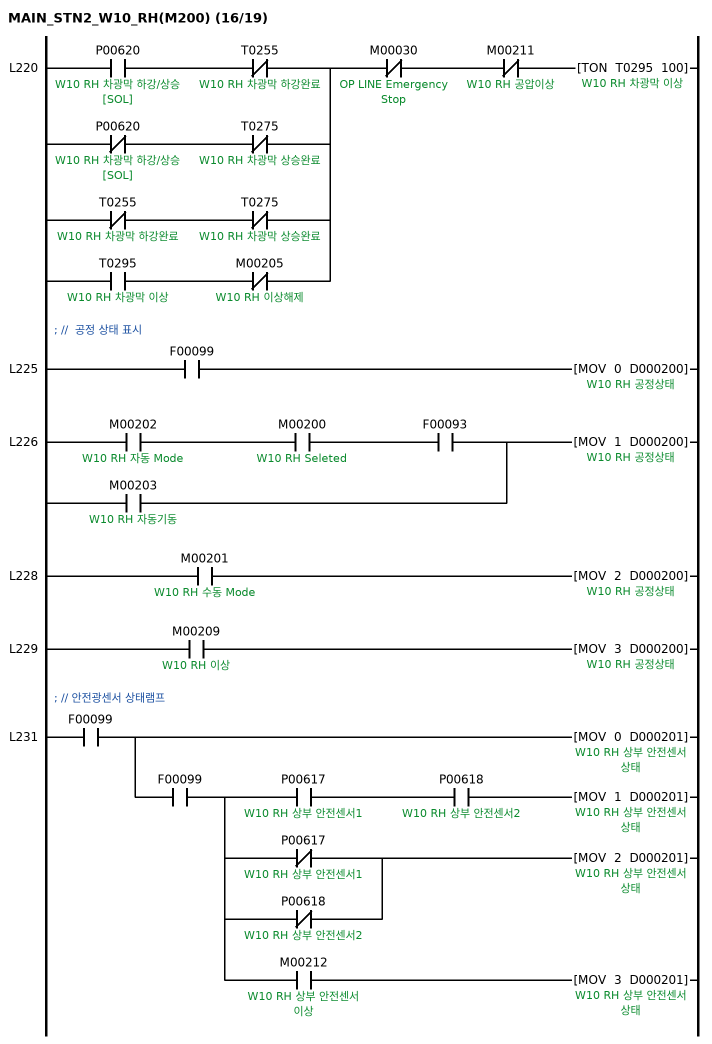
[picture p72: MAIN_STN2_W10_RH(M200) rungs L220-L231]
; L220
LOAD      P00620	// W10 RH 차광막 하강/상승 [SOL]
AND NOT   T0255	// W10 RH 차광막 하강완료
LOAD NOT  P00620	// W10 RH 차광막 하강/상승 [SOL]
AND NOT   T0275	// W10 RH 차광막 상승완료
OR LOAD
LOAD NOT  T0255	// W10 RH 차광막 하강완료
AND NOT   T0275	// W10 RH 차광막 상승완료
OR LOAD
LOAD      T0295	// W10 RH 차광막 이상
AND NOT   M00205	// W10 RH 이상해제
OR LOAD
AND NOT   M00030	// OP LINE Emergency Stop
AND NOT   M00211	// W10 RH 공압이상
TON       T0295 100	// W10 RH 차광막 이상
//   //  공정 상태 표시
; L225
LOAD      F00099
MOV       0 D000200	// W10 RH 공정상태
; L226
LOAD      M00202	// W10 RH 자동 Mode
AND       M00200	// W10 RH Seleted
AND       F00093
OR        M00203	// W10 RH 자동기동
MOV       1 D000200	// W10 RH 공정상태
; L228
LOAD      M00201	// W10 RH 수동 Mode
MOV       2 D000200	// W10 RH 공정상태
; L229
LOAD      M00209	// W10 RH 이상
MOV       3 D000200	// W10 RH 공정상태
//   // 안전광센서 상태램프
; L231
LOAD      F00099
MOV       0 D000201	// W10 RH 상부 안전센서 상태
AND       F00099
MPUSH
AND       P00617	// W10 RH 상부 안전센서1
AND       P00618	// W10 RH 상부 안전센서2
MOV       1 D000201	// W10 RH 상부 안전센서 상태
MLOAD
LOAD NOT  P00617	// W10 RH 상부 안전센서1
OR NOT    P00618	// W10 RH 상부 안전센서2
AND LOAD
MOV       2 D000201	// W10 RH 상부 안전센서 상태
MPOP
AND       M00212	// W10 RH 상부 안전센서 이상
MOV       3 D000201	// W10 RH 상부 안전센서 상태

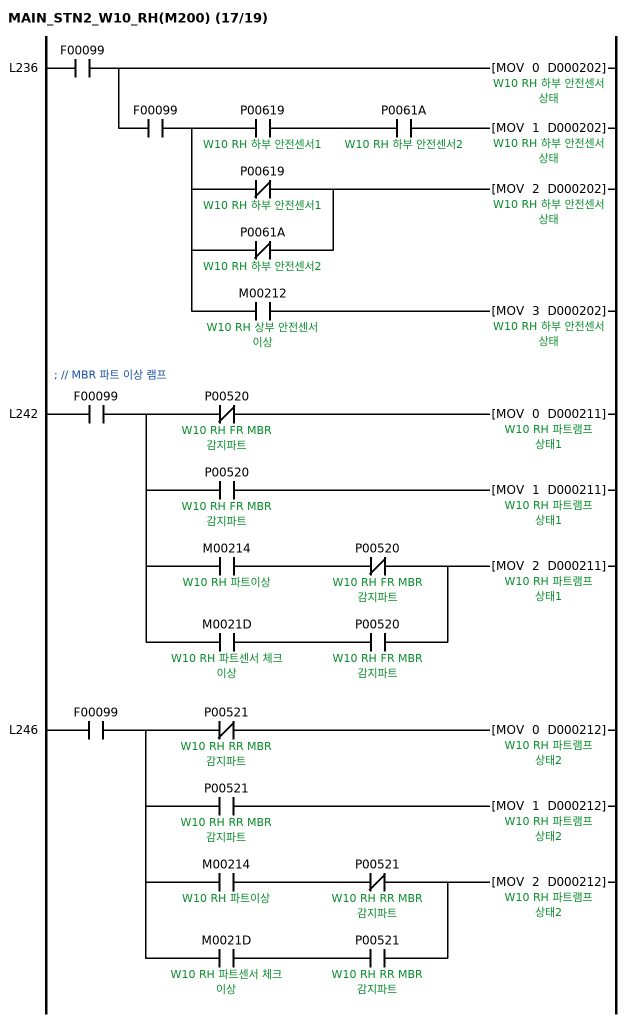
; L236
LOAD      F00099
MOV       0 D000202	// W10 RH 하부 안전센서 상태
AND       F00099
MPUSH
AND       P00619	// W10 RH 하부 안전센서1
AND       P0061A	// W10 RH 하부 안전센서2
MOV       1 D000202	// W10 RH 하부 안전센서 상태
MLOAD
LOAD NOT  P00619	// W10 RH 하부 안전센서1
OR NOT    P0061A	// W10 RH 하부 안전센서2
AND LOAD
MOV       2 D000202	// W10 RH 하부 안전센서 상태
MPOP
AND       M00212	// W10 RH 상부 안전센서 이상
MOV       3 D000202	// W10 RH 하부 안전센서 상태
//   // MBR 파트 이상 램프
; L242
LOAD      F00099
MPUSH
AND NOT   P00520	// W10 RH FR MBR 감지파트
MOV       0 D000211	// W10 RH 파트램프 상태1
MLOAD
AND       P00520	// W10 RH FR MBR 감지파트
MOV       1 D000211	// W10 RH 파트램프 상태1
MPOP
LOAD      M00214	// W10 RH 파트이상
AND NOT   P00520	// W10 RH FR MBR 감지파트
LOAD      M0021D	// W10 RH 파트센서 체크 이상
AND       P00520	// W10 RH FR MBR 감지파트
OR LOAD
AND LOAD
MOV       2 D000211	// W10 RH 파트램프 상태1
; L246
LOAD      F00099
MPUSH
AND NOT   P00521	// W10 RH RR MBR 감지파트
MOV       0 D000212	// W10 RH 파트램프 상태2
MLOAD
AND       P00521	// W10 RH RR MBR 감지파트
MOV       1 D000212	// W10 RH 파트램프 상태2
MPOP
LOAD      M00214	// W10 RH 파트이상
AND NOT   P00521	// W10 RH RR MBR 감지파트
LOAD      M0021D	// W10 RH 파트센서 체크 이상
AND       P00521	// W10 RH RR MBR 감지파트
OR LOAD
AND LOAD
MOV       2 D000212	// W10 RH 파트램프 상태2

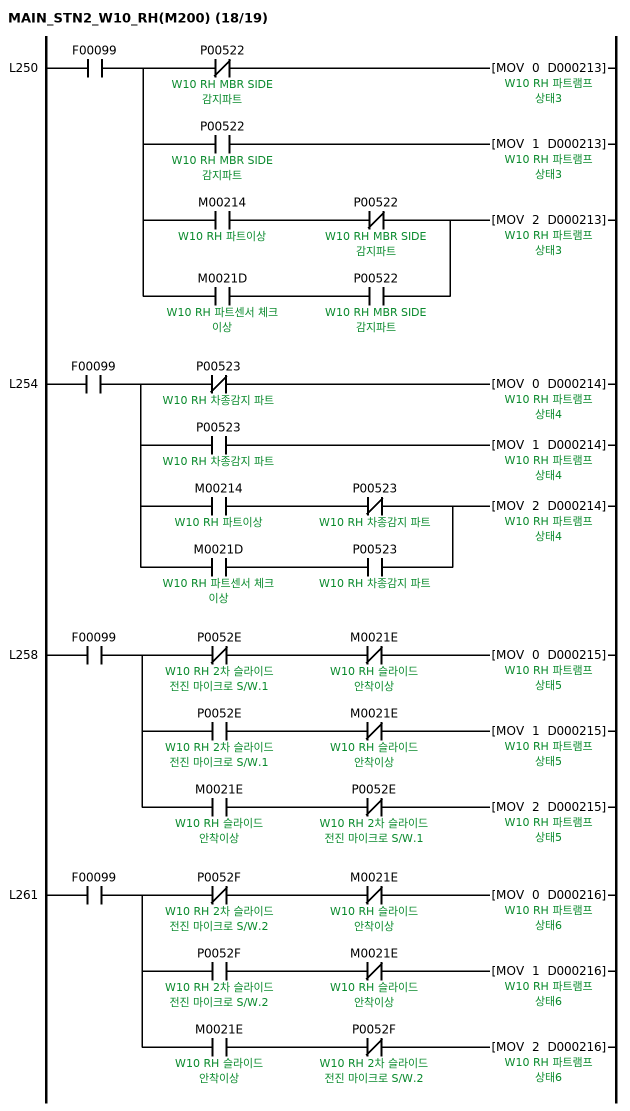
; L250
LOAD      F00099
MPUSH
AND NOT   P00522	// W10 RH MBR SIDE 감지파트
MOV       0 D000213	// W10 RH 파트램프 상태3
MLOAD
AND       P00522	// W10 RH MBR SIDE 감지파트
MOV       1 D000213	// W10 RH 파트램프 상태3
MPOP
LOAD      M00214	// W10 RH 파트이상
AND NOT   P00522	// W10 RH MBR SIDE 감지파트
LOAD      M0021D	// W10 RH 파트센서 체크 이상
AND       P00522	// W10 RH MBR SIDE 감지파트
OR LOAD
AND LOAD
MOV       2 D000213	// W10 RH 파트램프 상태3
; L254
LOAD      F00099
MPUSH
AND NOT   P00523	// W10 RH 차종감지 파트
MOV       0 D000214	// W10 RH 파트램프 상태4
MLOAD
AND       P00523	// W10 RH 차종감지 파트
MOV       1 D000214	// W10 RH 파트램프 상태4
MPOP
LOAD      M00214	// W10 RH 파트이상
AND NOT   P00523	// W10 RH 차종감지 파트
LOAD      M0021D	// W10 RH 파트센서 체크 이상
AND       P00523	// W10 RH 차종감지 파트
OR LOAD
AND LOAD
MOV       2 D000214	// W10 RH 파트램프 상태4
; L258
LOAD      F00099
MPUSH
AND NOT   P0052E	// W10 RH 2차 슬라이드 전진 마이크로 S/W.1
AND NOT   M0021E	// W10 RH 슬라이드 안착이상
MOV       0 D000215	// W10 RH 파트램프 상태5
MLOAD
AND       P0052E	// W10 RH 2차 슬라이드 전진 마이크로 S/W.1
AND NOT   M0021E	// W10 RH 슬라이드 안착이상
MOV       1 D000215	// W10 RH 파트램프 상태5
MPOP
AND       M0021E	// W10 RH 슬라이드 안착이상
AND NOT   P0052E	// W10 RH 2차 슬라이드 전진 마이크로 S/W.1
MOV       2 D000215	// W10 RH 파트램프 상태5
; L261
LOAD      F00099
MPUSH
AND NOT   P0052F	// W10 RH 2차 슬라이드 전진 마이크로 S/W.2
AND NOT   M0021E	// W10 RH 슬라이드 안착이상
MOV       0 D000216	// W10 RH 파트램프 상태6
MLOAD
AND       P0052F	// W10 RH 2차 슬라이드 전진 마이크로 S/W.2
AND NOT   M0021E	// W10 RH 슬라이드 안착이상
MOV       1 D000216	// W10 RH 파트램프 상태6
MPOP
AND       M0021E	// W10 RH 슬라이드 안착이상
AND NOT   P0052F	// W10 RH 2차 슬라이드 전진 마이크로 S/W.2
MOV       2 D000216	// W10 RH 파트램프 상태6

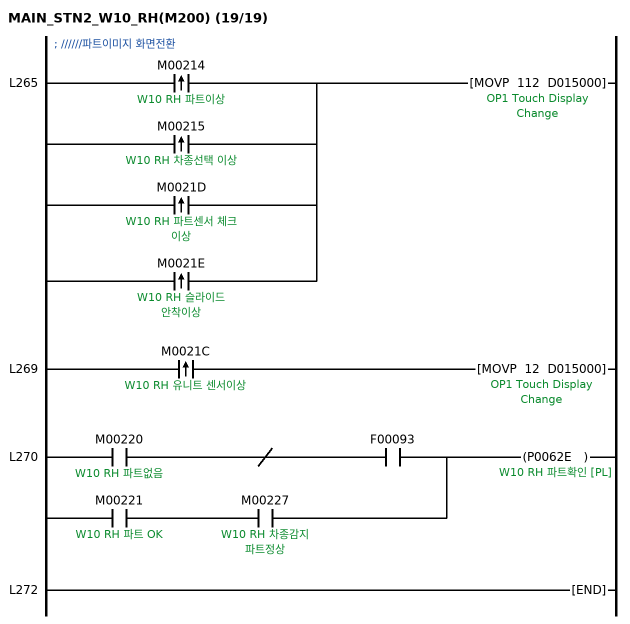
// //////파트이미지 화면전환
; L265
LOADP     M00214	// W10 RH 파트이상
ORP       M00215	// W10 RH 차종선택 이상
ORP       M0021D	// W10 RH 파트센서 체크 이상
ORP       M0021E	// W10 RH 슬라이드 안착이상
MOVP      112 D015000	// OP1 Touch Display Change
; L269
LOADP     M0021C	// W10 RH 유니트 센서이상
MOVP      12 D015000	// OP1 Touch Display Change
; L270
LOAD      M00220	// W10 RH 파트없음
NOT
AND       F00093
LOAD      M00221	// W10 RH 파트 OK
AND       M00227	// W10 RH 차종감지 파트정상
OR LOAD
OUT       P0062E	// W10 RH 파트확인 [PL]
; L272
END

PROGRAM MAIN_STN3_W20_LH_냉각(M300) (task: 스캔 프로그램)

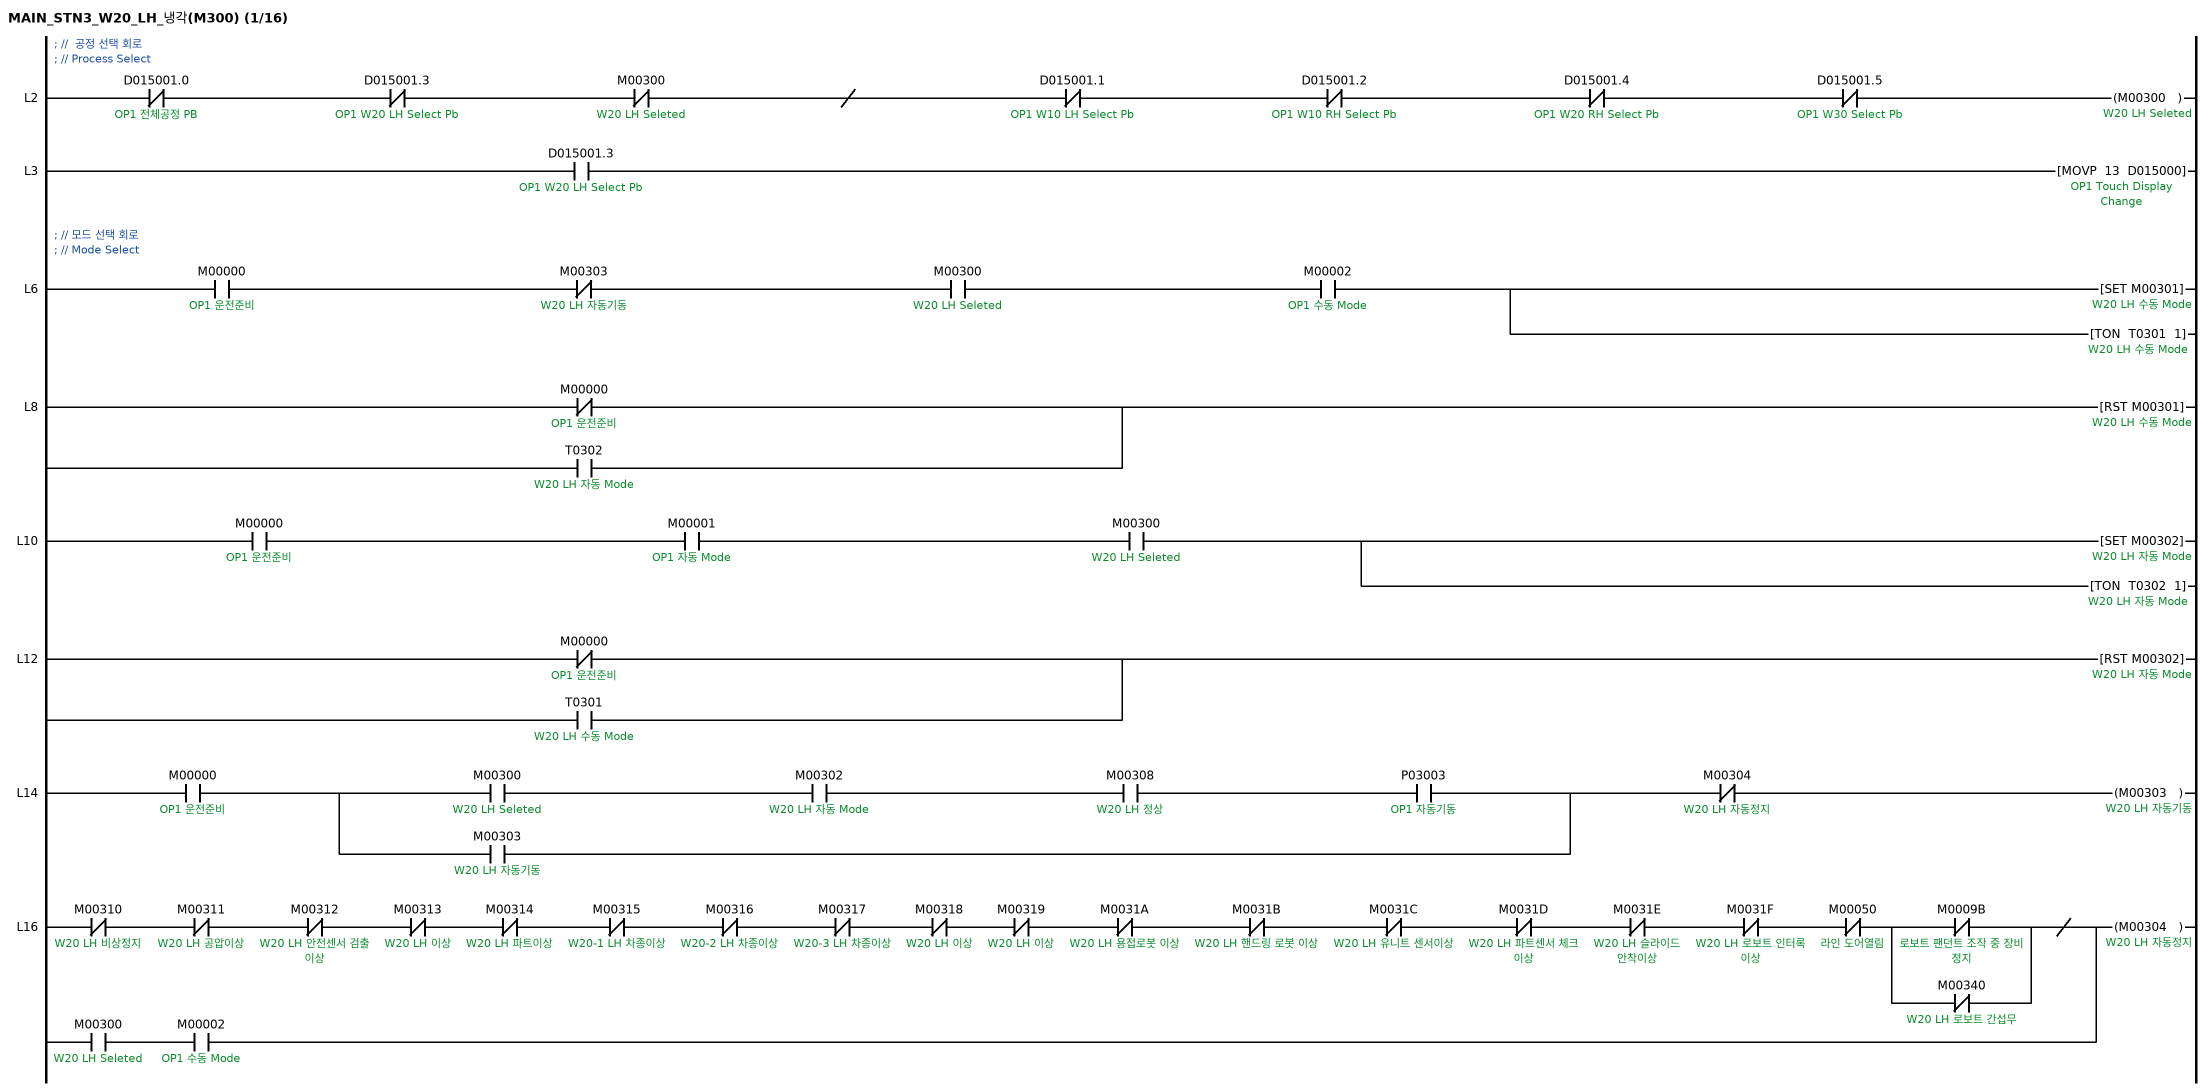
//   //  공정 선택 회로
//   // Process Select
; L2
LOAD NOT  D015001.0	// OP1 전체공정 PB
AND NOT   D015001.3	// OP1 W20 LH Select Pb
AND NOT   M00300	// W20 LH Seleted
NOT
AND NOT   D015001.1	// OP1 W10 LH Select Pb
AND NOT   D015001.2	// OP1 W10 RH Select Pb
AND NOT   D015001.4	// OP1 W20 RH Select Pb
AND NOT   D015001.5	// OP1 W30 Select Pb
OUT       M00300	// W20 LH Seleted
; L3
LOAD      D015001.3	// OP1 W20 LH Select Pb
MOVP      13 D015000	// OP1 Touch Display Change
// // 모드 선택 회로
//   // Mode Select
; L6
LOAD      M00000	// OP1 운전준비
AND NOT   M00303	// W20 LH 자동기동
AND       M00300	// W20 LH Seleted
AND       M00002	// OP1 수동 Mode
SET       M00301	// W20 LH 수동 Mode
TON       T0301 1	// W20 LH 수동 Mode
; L8
LOAD NOT  M00000	// OP1 운전준비
OR        T0302	// W20 LH 자동 Mode
RST       M00301	// W20 LH 수동 Mode
; L10
LOAD      M00000	// OP1 운전준비
AND       M00001	// OP1 자동 Mode
AND       M00300	// W20 LH Seleted
SET       M00302	// W20 LH 자동 Mode
TON       T0302 1	// W20 LH 자동 Mode
; L12
LOAD NOT  M00000	// OP1 운전준비
OR        T0301	// W20 LH 수동 Mode
RST       M00302	// W20 LH 자동 Mode
; L14
LOAD      M00000	// OP1 운전준비
LOAD      M00300	// W20 LH Seleted
AND       M00302	// W20 LH 자동 Mode
AND       M00308	// W20 LH 정상
AND       P03003	// OP1 자동기동
OR        M00303	// W20 LH 자동기동
AND LOAD
AND NOT   M00304	// W20 LH 자동정지
OUT       M00303	// W20 LH 자동기동
; L16
LOAD NOT  M00310	// W20 LH 비상정지
AND NOT   M00311	// W20 LH 공압이상
AND NOT   M00312	// W20 LH 안전센서 검출 이상
AND NOT   M00313	// W20 LH 이상
AND NOT   M00314	// W20 LH 파트이상
AND NOT   M00315	// W20-1 LH 차종이상
AND NOT   M00316	// W20-2 LH 차종이상
AND NOT   M00317	// W20-3 LH 차종이상
AND NOT   M00318	// W20 LH 이상
AND NOT   M00319	// W20 LH 이상
AND NOT   M0031A	// W20 LH 용접로봇 이상
AND NOT   M0031B	// W20 LH 핸드링 로봇 이상
AND NOT   M0031C	// W20 LH 유니트 센서이상
AND NOT   M0031D	// W20 LH 파트센서 체크 이상
AND NOT   M0031E	// W20 LH 슬라이드 안착이상
AND NOT   M0031F	// W20 LH 로보트 인터록 이상
AND NOT   M00050	// 라인 도어열림
LOAD NOT  M0009B	// 로보트 팬던트 조작 중 장비 정지
OR NOT    M00340	// W20 LH 로보트 간섭무
AND LOAD
NOT
LOAD      M00300	// W20 LH Seleted
AND       M00002	// OP1 수동 Mode
OR LOAD
OUT       M00304	// W20 LH 자동정지

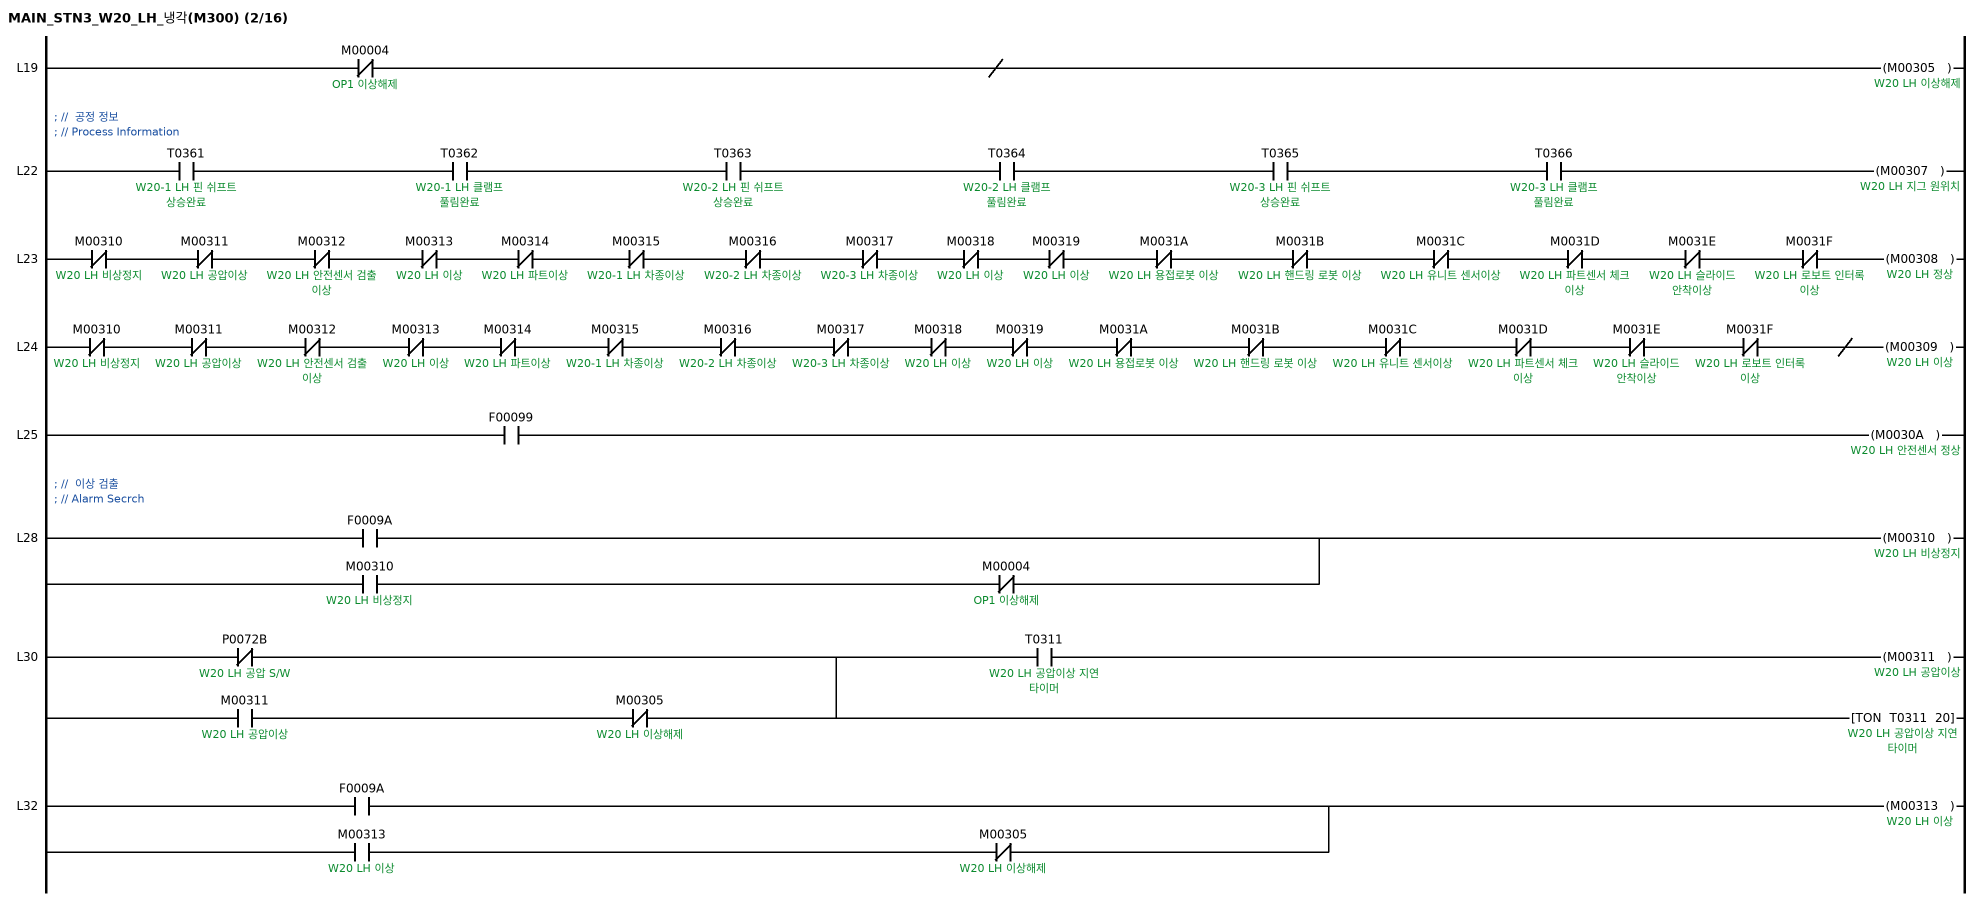
; L19
LOAD NOT  M00004	// OP1 이상해제
NOT
OUT       M00305	// W20 LH 이상해제
//   //  공정 정보
//   // Process Information
; L22
LOAD      T0361	// W20-1 LH 핀 쉬프트 상승완료
AND       T0362	// W20-1 LH 클램프 풀림완료
AND       T0363	// W20-2 LH 핀 쉬프트 상승완료
AND       T0364	// W20-2 LH 클램프 풀림완료
AND       T0365	// W20-3 LH 핀 쉬프트 상승완료
AND       T0366	// W20-3 LH 클램프 풀림완료
OUT       M00307	// W20 LH 지그 원위치
; L23
LOAD NOT  M00310	// W20 LH 비상정지
AND NOT   M00311	// W20 LH 공압이상
AND NOT   M00312	// W20 LH 안전센서 검출 이상
AND NOT   M00313	// W20 LH 이상
AND NOT   M00314	// W20 LH 파트이상
AND NOT   M00315	// W20-1 LH 차종이상
AND NOT   M00316	// W20-2 LH 차종이상
AND NOT   M00317	// W20-3 LH 차종이상
AND NOT   M00318	// W20 LH 이상
AND NOT   M00319	// W20 LH 이상
AND NOT   M0031A	// W20 LH 용접로봇 이상
AND NOT   M0031B	// W20 LH 핸드링 로봇 이상
AND NOT   M0031C	// W20 LH 유니트 센서이상
AND NOT   M0031D	// W20 LH 파트센서 체크 이상
AND NOT   M0031E	// W20 LH 슬라이드 안착이상
AND NOT   M0031F	// W20 LH 로보트 인터록 이상
OUT       M00308	// W20 LH 정상
; L24
LOAD NOT  M00310	// W20 LH 비상정지
AND NOT   M00311	// W20 LH 공압이상
AND NOT   M00312	// W20 LH 안전센서 검출 이상
AND NOT   M00313	// W20 LH 이상
AND NOT   M00314	// W20 LH 파트이상
AND NOT   M00315	// W20-1 LH 차종이상
AND NOT   M00316	// W20-2 LH 차종이상
AND NOT   M00317	// W20-3 LH 차종이상
AND NOT   M00318	// W20 LH 이상
AND NOT   M00319	// W20 LH 이상
AND NOT   M0031A	// W20 LH 용접로봇 이상
AND NOT   M0031B	// W20 LH 핸드링 로봇 이상
AND NOT   M0031C	// W20 LH 유니트 센서이상
AND NOT   M0031D	// W20 LH 파트센서 체크 이상
AND NOT   M0031E	// W20 LH 슬라이드 안착이상
AND NOT   M0031F	// W20 LH 로보트 인터록 이상
NOT
OUT       M00309	// W20 LH 이상
; L25
LOAD      F00099
OUT       M0030A	// W20 LH 안전센서 정상
//   //  이상 검출
//   // Alarm Secrch
; L28
LOAD      F0009A
LOAD      M00310	// W20 LH 비상정지
AND NOT   M00004	// OP1 이상해제
OR LOAD
OUT       M00310	// W20 LH 비상정지
; L30
LOAD NOT  P0072B	// W20 LH 공압 S/W
LOAD      M00311	// W20 LH 공압이상
AND NOT   M00305	// W20 LH 이상해제
OR LOAD
MPUSH
AND       T0311	// W20 LH 공압이상 지연 타이머
OUT       M00311	// W20 LH 공압이상
MPOP
TON       T0311 20	// W20 LH 공압이상 지연 타이머
; L32
LOAD      F0009A
LOAD      M00313	// W20 LH 이상
AND NOT   M00305	// W20 LH 이상해제
OR LOAD
OUT       M00313	// W20 LH 이상

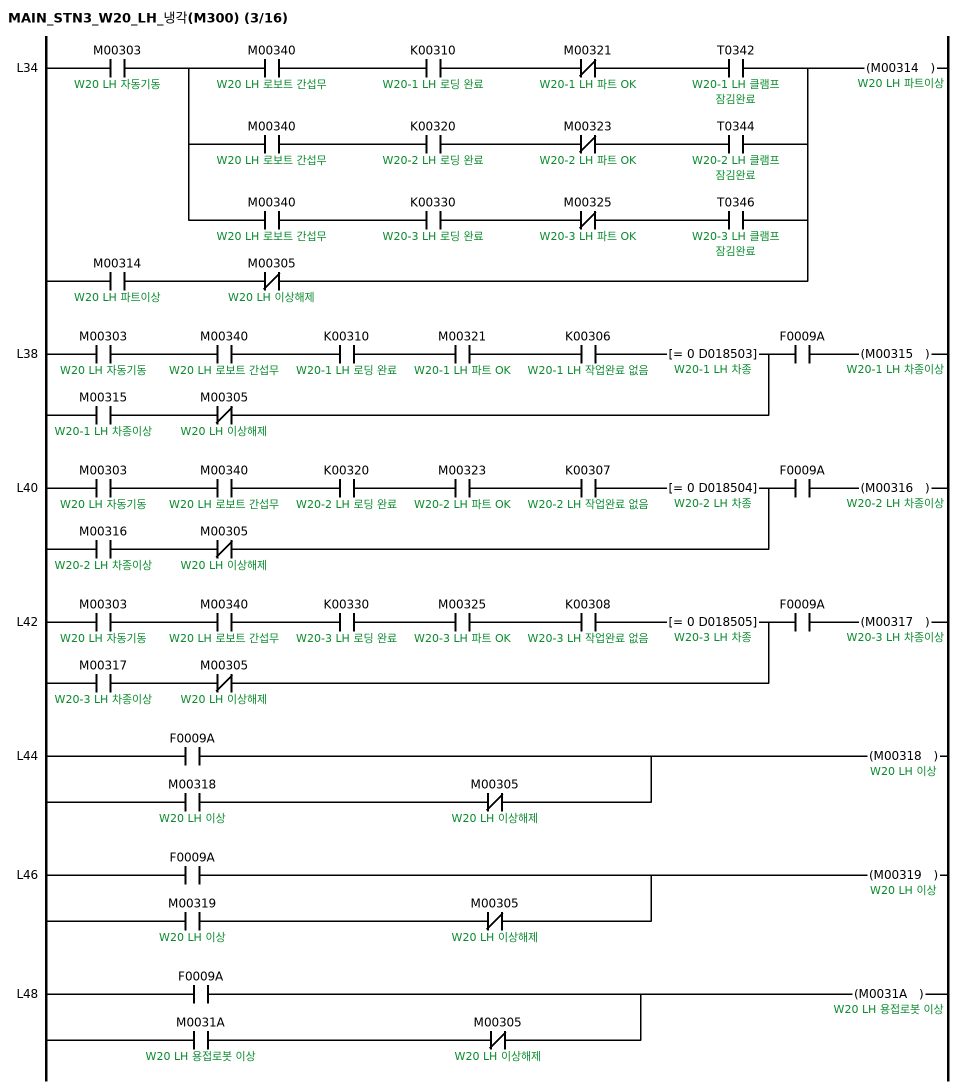
; L34
LOAD      M00303	// W20 LH 자동기동
LOAD      M00340	// W20 LH 로보트 간섭무
AND       K00310	// W20-1 LH 로딩 완료
AND NOT   M00321	// W20-1 LH 파트 OK
AND       T0342	// W20-1 LH 클램프 잠김완료
LOAD      M00340	// W20 LH 로보트 간섭무
AND       K00320	// W20-2 LH 로딩 완료
AND NOT   M00323	// W20-2 LH 파트 OK
AND       T0344	// W20-2 LH 클램프 잠김완료
OR LOAD
LOAD      M00340	// W20 LH 로보트 간섭무
AND       K00330	// W20-3 LH 로딩 완료
AND NOT   M00325	// W20-3 LH 파트 OK
AND       T0346	// W20-3 LH 클램프 잠김완료
OR LOAD
AND LOAD
LOAD      M00314	// W20 LH 파트이상
AND NOT   M00305	// W20 LH 이상해제
OR LOAD
OUT       M00314	// W20 LH 파트이상
; L38
LOAD      M00303	// W20 LH 자동기동
AND       M00340	// W20 LH 로보트 간섭무
AND       K00310	// W20-1 LH 로딩 완료
AND       M00321	// W20-1 LH 파트 OK
AND       K00306	// W20-1 LH 작업완료 없음
AND=      0 D018503	// W20-1 LH 차종
LOAD      M00315	// W20-1 LH 차종이상
AND NOT   M00305	// W20 LH 이상해제
OR LOAD
AND       F0009A
OUT       M00315	// W20-1 LH 차종이상
; L40
LOAD      M00303	// W20 LH 자동기동
AND       M00340	// W20 LH 로보트 간섭무
AND       K00320	// W20-2 LH 로딩 완료
AND       M00323	// W20-2 LH 파트 OK
AND       K00307	// W20-2 LH 작업완료 없음
AND=      0 D018504	// W20-2 LH 차종
LOAD      M00316	// W20-2 LH 차종이상
AND NOT   M00305	// W20 LH 이상해제
OR LOAD
AND       F0009A
OUT       M00316	// W20-2 LH 차종이상
; L42
LOAD      M00303	// W20 LH 자동기동
AND       M00340	// W20 LH 로보트 간섭무
AND       K00330	// W20-3 LH 로딩 완료
AND       M00325	// W20-3 LH 파트 OK
AND       K00308	// W20-3 LH 작업완료 없음
AND=      0 D018505	// W20-3 LH 차종
LOAD      M00317	// W20-3 LH 차종이상
AND NOT   M00305	// W20 LH 이상해제
OR LOAD
AND       F0009A
OUT       M00317	// W20-3 LH 차종이상
; L44
LOAD      F0009A
LOAD      M00318	// W20 LH 이상
AND NOT   M00305	// W20 LH 이상해제
OR LOAD
OUT       M00318	// W20 LH 이상
; L46
LOAD      F0009A
LOAD      M00319	// W20 LH 이상
AND NOT   M00305	// W20 LH 이상해제
OR LOAD
OUT       M00319	// W20 LH 이상
; L48
LOAD      F0009A
LOAD      M0031A	// W20 LH 용접로봇 이상
AND NOT   M00305	// W20 LH 이상해제
OR LOAD
OUT       M0031A	// W20 LH 용접로봇 이상

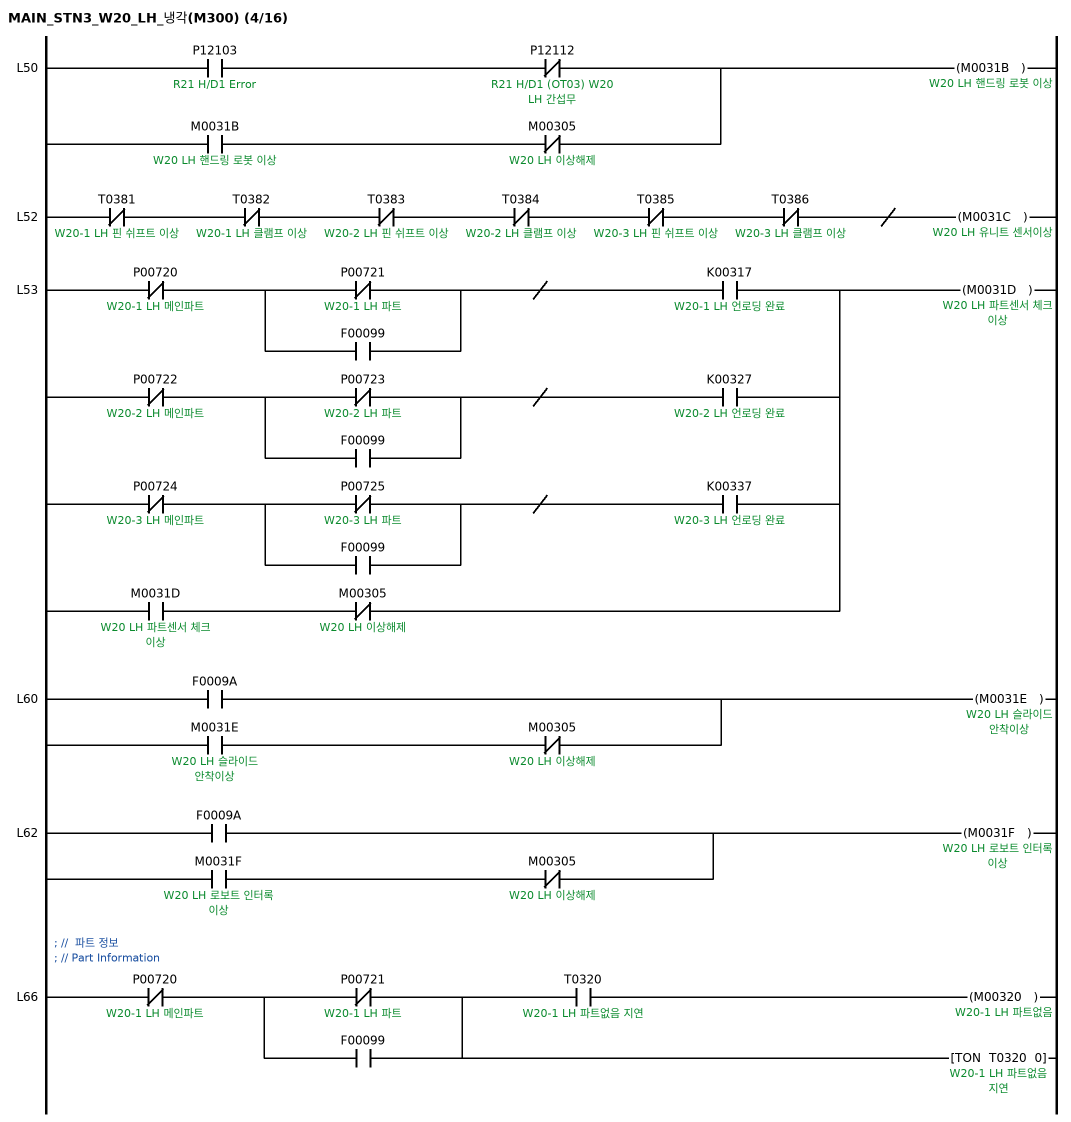
; L50
LOAD      P12103	// R21 H/D1 Error
AND NOT   P12112	// R21 H/D1 (OT03) W20 LH 간섭무
LOAD      M0031B	// W20 LH 핸드링 로봇 이상
AND NOT   M00305	// W20 LH 이상해제
OR LOAD
OUT       M0031B	// W20 LH 핸드링 로봇 이상
; L52
LOAD NOT  T0381	// W20-1 LH 핀 쉬프트 이상
AND NOT   T0382	// W20-1 LH 클램프 이상
AND NOT   T0383	// W20-2 LH 핀 쉬프트 이상
AND NOT   T0384	// W20-2 LH 클램프 이상
AND NOT   T0385	// W20-3 LH 핀 쉬프트 이상
AND NOT   T0386	// W20-3 LH 클램프 이상
NOT
OUT       M0031C	// W20 LH 유니트 센서이상
; L53
LOAD NOT  P00720	// W20-1 LH 메인파트
LOAD NOT  P00721	// W20-1 LH 파트
OR        F00099
AND LOAD
NOT
AND       K00317	// W20-1 LH 언로딩 완료
LOAD NOT  P00722	// W20-2 LH 메인파트
LOAD NOT  P00723	// W20-2 LH 파트
OR        F00099
AND LOAD
NOT
AND       K00327	// W20-2 LH 언로딩 완료
OR LOAD
LOAD NOT  P00724	// W20-3 LH 메인파트
LOAD NOT  P00725	// W20-3 LH 파트
OR        F00099
AND LOAD
NOT
AND       K00337	// W20-3 LH 언로딩 완료
OR LOAD
LOAD      M0031D	// W20 LH 파트센서 체크 이상
AND NOT   M00305	// W20 LH 이상해제
OR LOAD
OUT       M0031D	// W20 LH 파트센서 체크 이상
; L60
LOAD      F0009A
LOAD      M0031E	// W20 LH 슬라이드 안착이상
AND NOT   M00305	// W20 LH 이상해제
OR LOAD
OUT       M0031E	// W20 LH 슬라이드 안착이상
; L62
LOAD      F0009A
LOAD      M0031F	// W20 LH 로보트 인터록 이상
AND NOT   M00305	// W20 LH 이상해제
OR LOAD
OUT       M0031F	// W20 LH 로보트 인터록 이상
//   //  파트 정보
//   // Part Information
; L66
LOAD NOT  P00720	// W20-1 LH 메인파트
LOAD NOT  P00721	// W20-1 LH 파트
OR        F00099
AND LOAD
MPUSH
AND       T0320	// W20-1 LH 파트없음 지연
OUT       M00320	// W20-1 LH 파트없음
MPOP
TON       T0320 0	// W20-1 LH 파트없음 지연

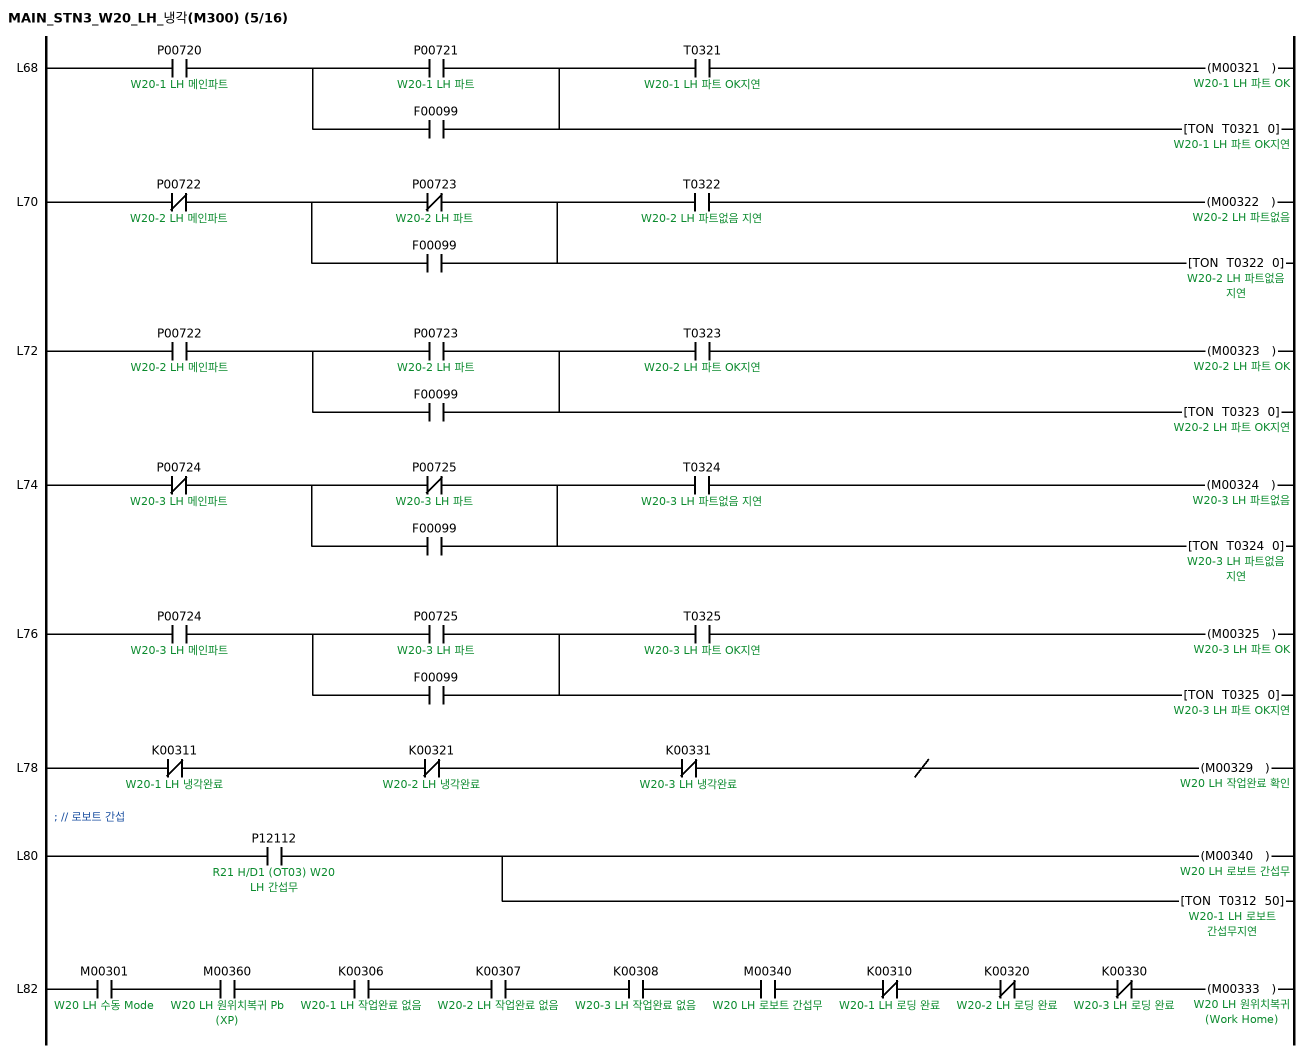
; L68
LOAD      P00720	// W20-1 LH 메인파트
LOAD      P00721	// W20-1 LH 파트
OR        F00099
AND LOAD
MPUSH
AND       T0321	// W20-1 LH 파트 OK지연
OUT       M00321	// W20-1 LH 파트 OK
MPOP
TON       T0321 0	// W20-1 LH 파트 OK지연
; L70
LOAD NOT  P00722	// W20-2 LH 메인파트
LOAD NOT  P00723	// W20-2 LH 파트
OR        F00099
AND LOAD
MPUSH
AND       T0322	// W20-2 LH 파트없음 지연
OUT       M00322	// W20-2 LH 파트없음
MPOP
TON       T0322 0	// W20-2 LH 파트없음 지연
; L72
LOAD      P00722	// W20-2 LH 메인파트
LOAD      P00723	// W20-2 LH 파트
OR        F00099
AND LOAD
MPUSH
AND       T0323	// W20-2 LH 파트 OK지연
OUT       M00323	// W20-2 LH 파트 OK
MPOP
TON       T0323 0	// W20-2 LH 파트 OK지연
; L74
LOAD NOT  P00724	// W20-3 LH 메인파트
LOAD NOT  P00725	// W20-3 LH 파트
OR        F00099
AND LOAD
MPUSH
AND       T0324	// W20-3 LH 파트없음 지연
OUT       M00324	// W20-3 LH 파트없음
MPOP
TON       T0324 0	// W20-3 LH 파트없음 지연
; L76
LOAD      P00724	// W20-3 LH 메인파트
LOAD      P00725	// W20-3 LH 파트
OR        F00099
AND LOAD
MPUSH
AND       T0325	// W20-3 LH 파트 OK지연
OUT       M00325	// W20-3 LH 파트 OK
MPOP
TON       T0325 0	// W20-3 LH 파트 OK지연
; L78
LOAD NOT  K00311	// W20-1 LH 냉각완료
AND NOT   K00321	// W20-2 LH 냉각완료
AND NOT   K00331	// W20-3 LH 냉각완료
NOT
OUT       M00329	// W20 LH 작업완료 확인
//   // 로보트 간섭
; L80
LOAD      P12112	// R21 H/D1 (OT03) W20 LH 간섭무
OUT       M00340	// W20 LH 로보트 간섭무
TON       T0312 50	// W20-1 LH 로보트 간섭무지연
; L82
LOAD      M00301	// W20 LH 수동 Mode
AND       M00360	// W20 LH 원위치복귀 Pb (XP)
AND       K00306	// W20-1 LH 작업완료 없음
AND       K00307	// W20-2 LH 작업완료 없음
AND       K00308	// W20-3 LH 작업완료 없음
AND       M00340	// W20 LH 로보트 간섭무
AND NOT   K00310	// W20-1 LH 로딩 완료
AND NOT   K00320	// W20-2 LH 로딩 완료
AND NOT   K00330	// W20-3 LH 로딩 완료
OUT       M00333	// W20 LH 원위치복귀 (Work Home)

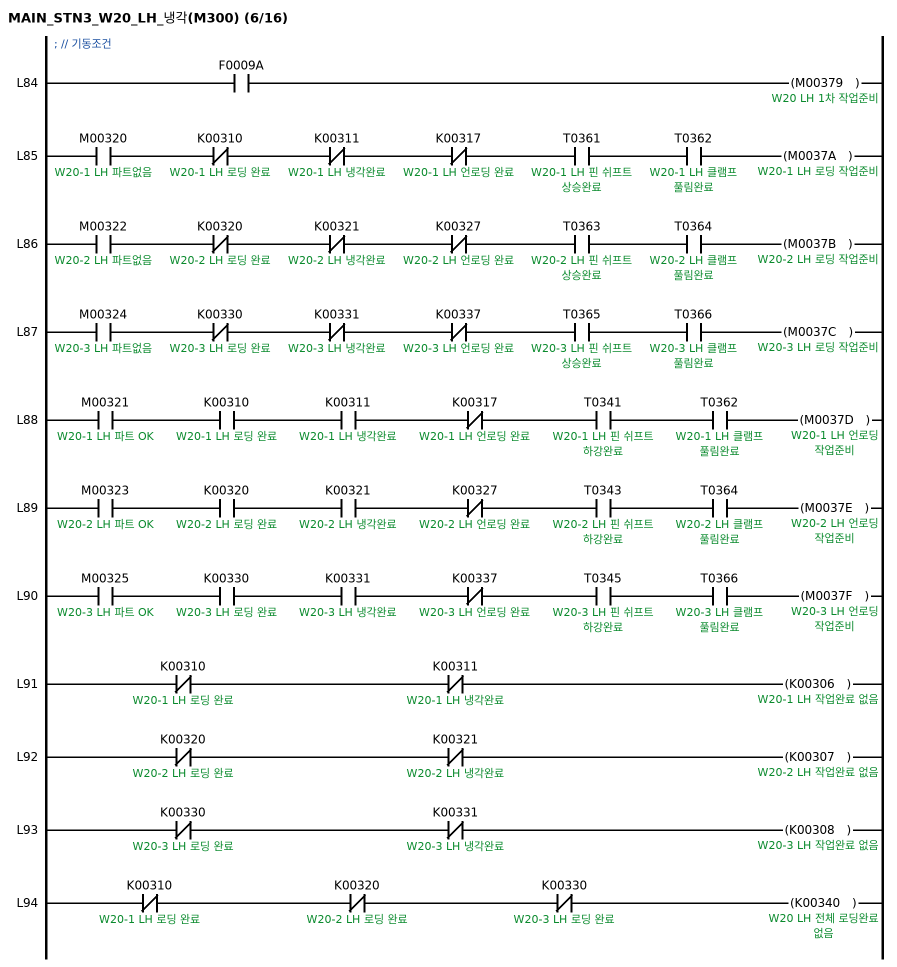
//   // 기동조건
; L84
LOAD      F0009A
OUT       M00379	// W20 LH 1차 작업준비
; L85
LOAD      M00320	// W20-1 LH 파트없음
AND NOT   K00310	// W20-1 LH 로딩 완료
AND NOT   K00311	// W20-1 LH 냉각완료
AND NOT   K00317	// W20-1 LH 언로딩 완료
AND       T0361	// W20-1 LH 핀 쉬프트 상승완료
AND       T0362	// W20-1 LH 클램프 풀림완료
OUT       M0037A	// W20-1 LH 로딩 작업준비
; L86
LOAD      M00322	// W20-2 LH 파트없음
AND NOT   K00320	// W20-2 LH 로딩 완료
AND NOT   K00321	// W20-2 LH 냉각완료
AND NOT   K00327	// W20-2 LH 언로딩 완료
AND       T0363	// W20-2 LH 핀 쉬프트 상승완료
AND       T0364	// W20-2 LH 클램프 풀림완료
OUT       M0037B	// W20-2 LH 로딩 작업준비
; L87
LOAD      M00324	// W20-3 LH 파트없음
AND NOT   K00330	// W20-3 LH 로딩 완료
AND NOT   K00331	// W20-3 LH 냉각완료
AND NOT   K00337	// W20-3 LH 언로딩 완료
AND       T0365	// W20-3 LH 핀 쉬프트 상승완료
AND       T0366	// W20-3 LH 클램프 풀림완료
OUT       M0037C	// W20-3 LH 로딩 작업준비
; L88
LOAD      M00321	// W20-1 LH 파트 OK
AND       K00310	// W20-1 LH 로딩 완료
AND       K00311	// W20-1 LH 냉각완료
AND NOT   K00317	// W20-1 LH 언로딩 완료
AND       T0341	// W20-1 LH 핀 쉬프트 하강완료
AND       T0362	// W20-1 LH 클램프 풀림완료
OUT       M0037D	// W20-1 LH 언로딩 작업준비
; L89
LOAD      M00323	// W20-2 LH 파트 OK
AND       K00320	// W20-2 LH 로딩 완료
AND       K00321	// W20-2 LH 냉각완료
AND NOT   K00327	// W20-2 LH 언로딩 완료
AND       T0343	// W20-2 LH 핀 쉬프트 하강완료
AND       T0364	// W20-2 LH 클램프 풀림완료
OUT       M0037E	// W20-2 LH 언로딩 작업준비
; L90
LOAD      M00325	// W20-3 LH 파트 OK
AND       K00330	// W20-3 LH 로딩 완료
AND       K00331	// W20-3 LH 냉각완료
AND NOT   K00337	// W20-3 LH 언로딩 완료
AND       T0345	// W20-3 LH 핀 쉬프트 하강완료
AND       T0366	// W20-3 LH 클램프 풀림완료
OUT       M0037F	// W20-3 LH 언로딩 작업준비
; L91
LOAD NOT  K00310	// W20-1 LH 로딩 완료
AND NOT   K00311	// W20-1 LH 냉각완료
OUT       K00306	// W20-1 LH 작업완료 없음
; L92
LOAD NOT  K00320	// W20-2 LH 로딩 완료
AND NOT   K00321	// W20-2 LH 냉각완료
OUT       K00307	// W20-2 LH 작업완료 없음
; L93
LOAD NOT  K00330	// W20-3 LH 로딩 완료
AND NOT   K00331	// W20-3 LH 냉각완료
OUT       K00308	// W20-3 LH 작업완료 없음
; L94
LOAD NOT  K00310	// W20-1 LH 로딩 완료
AND NOT   K00320	// W20-2 LH 로딩 완료
AND NOT   K00330	// W20-3 LH 로딩 완료
OUT       K00340	// W20 LH 전체 로딩완료 없음

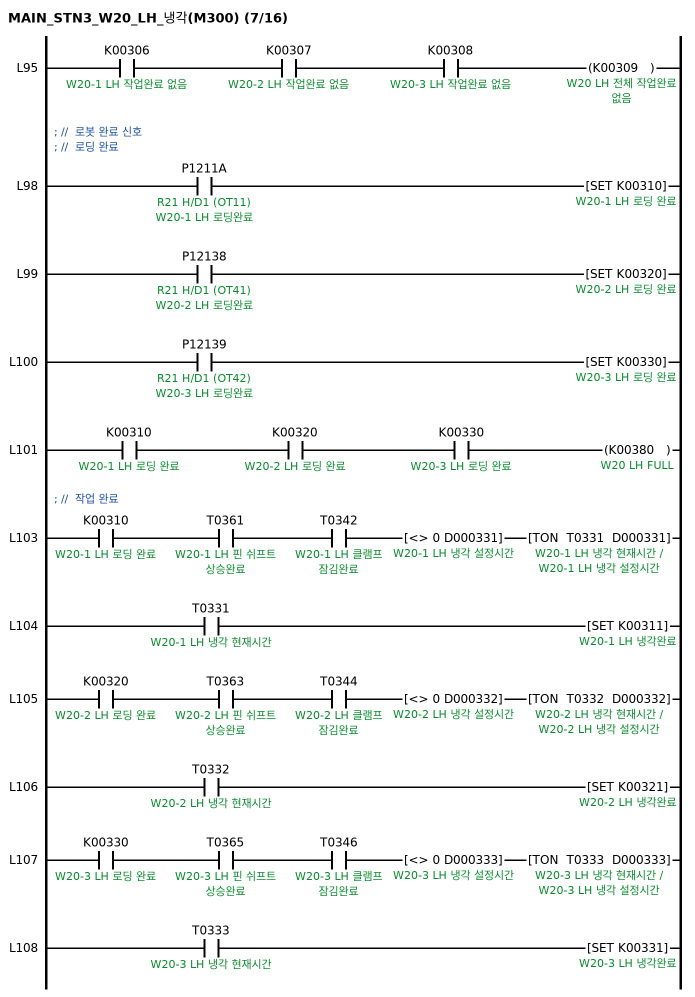
; L95
LOAD      K00306	// W20-1 LH 작업완료 없음
AND       K00307	// W20-2 LH 작업완료 없음
AND       K00308	// W20-3 LH 작업완료 없음
OUT       K00309	// W20 LH 전체 작업완료 없음
//   //  로봇 완료 신호
//   //  로딩 완료
; L98
LOAD      P1211A	// R21 H/D1 (OT11) W20-1 LH 로딩완료
SET       K00310	// W20-1 LH 로딩 완료
; L99
LOAD      P12138	// R21 H/D1 (OT41) W20-2 LH 로딩완료
SET       K00320	// W20-2 LH 로딩 완료
; L100
LOAD      P12139	// R21 H/D1 (OT42) W20-3 LH 로딩완료
SET       K00330	// W20-3 LH 로딩 완료
; L101
LOAD      K00310	// W20-1 LH 로딩 완료
AND       K00320	// W20-2 LH 로딩 완료
AND       K00330	// W20-3 LH 로딩 완료
OUT       K00380	// W20 LH FULL
//   //  작업 완료
; L103
LOAD      K00310	// W20-1 LH 로딩 완료
AND       T0361	// W20-1 LH 핀 쉬프트 상승완료
AND       T0342	// W20-1 LH 클램프 잠김완료
AND<>     0 D000331	// W20-1 LH 냉각 설정시간
TON       T0331 D000331	// W20-1 LH 냉각 현재시간 / W20-1 LH 냉각 설정시간
; L104
LOAD      T0331	// W20-1 LH 냉각 현재시간
SET       K00311	// W20-1 LH 냉각완료
; L105
LOAD      K00320	// W20-2 LH 로딩 완료
AND       T0363	// W20-2 LH 핀 쉬프트 상승완료
AND       T0344	// W20-2 LH 클램프 잠김완료
AND<>     0 D000332	// W20-2 LH 냉각 설정시간
TON       T0332 D000332	// W20-2 LH 냉각 현재시간 / W20-2 LH 냉각 설정시간
; L106
LOAD      T0332	// W20-2 LH 냉각 현재시간
SET       K00321	// W20-2 LH 냉각완료
; L107
LOAD      K00330	// W20-3 LH 로딩 완료
AND       T0365	// W20-3 LH 핀 쉬프트 상승완료
AND       T0346	// W20-3 LH 클램프 잠김완료
AND<>     0 D000333	// W20-3 LH 냉각 설정시간
TON       T0333 D000333	// W20-3 LH 냉각 현재시간 / W20-3 LH 냉각 설정시간
; L108
LOAD      T0333	// W20-3 LH 냉각 현재시간
SET       K00331	// W20-3 LH 냉각완료

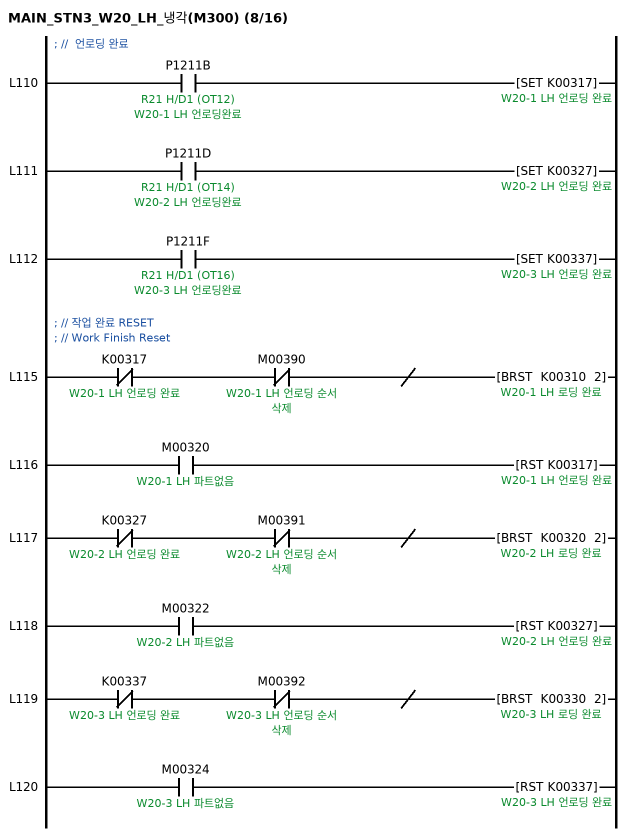
//   //  언로딩 완료
; L110
LOAD      P1211B	// R21 H/D1 (OT12) W20-1 LH 언로딩완료
SET       K00317	// W20-1 LH 언로딩 완료
; L111
LOAD      P1211D	// R21 H/D1 (OT14) W20-2 LH 언로딩완료
SET       K00327	// W20-2 LH 언로딩 완료
; L112
LOAD      P1211F	// R21 H/D1 (OT16) W20-3 LH 언로딩완료
SET       K00337	// W20-3 LH 언로딩 완료
//     // 작업 완료 RESET
//   // Work Finish Reset
; L115
LOAD NOT  K00317	// W20-1 LH 언로딩 완료
AND NOT   M00390	// W20-1 LH 언로딩 순서 삭제
NOT
BRST      K00310 2	// W20-1 LH 로딩 완료
; L116
LOAD      M00320	// W20-1 LH 파트없음
RST       K00317	// W20-1 LH 언로딩 완료
; L117
LOAD NOT  K00327	// W20-2 LH 언로딩 완료
AND NOT   M00391	// W20-2 LH 언로딩 순서 삭제
NOT
BRST      K00320 2	// W20-2 LH 로딩 완료
; L118
LOAD      M00322	// W20-2 LH 파트없음
RST       K00327	// W20-2 LH 언로딩 완료
; L119
LOAD NOT  K00337	// W20-3 LH 언로딩 완료
AND NOT   M00392	// W20-3 LH 언로딩 순서 삭제
NOT
BRST      K00330 2	// W20-3 LH 로딩 완료
; L120
LOAD      M00324	// W20-3 LH 파트없음
RST       K00337	// W20-3 LH 언로딩 완료

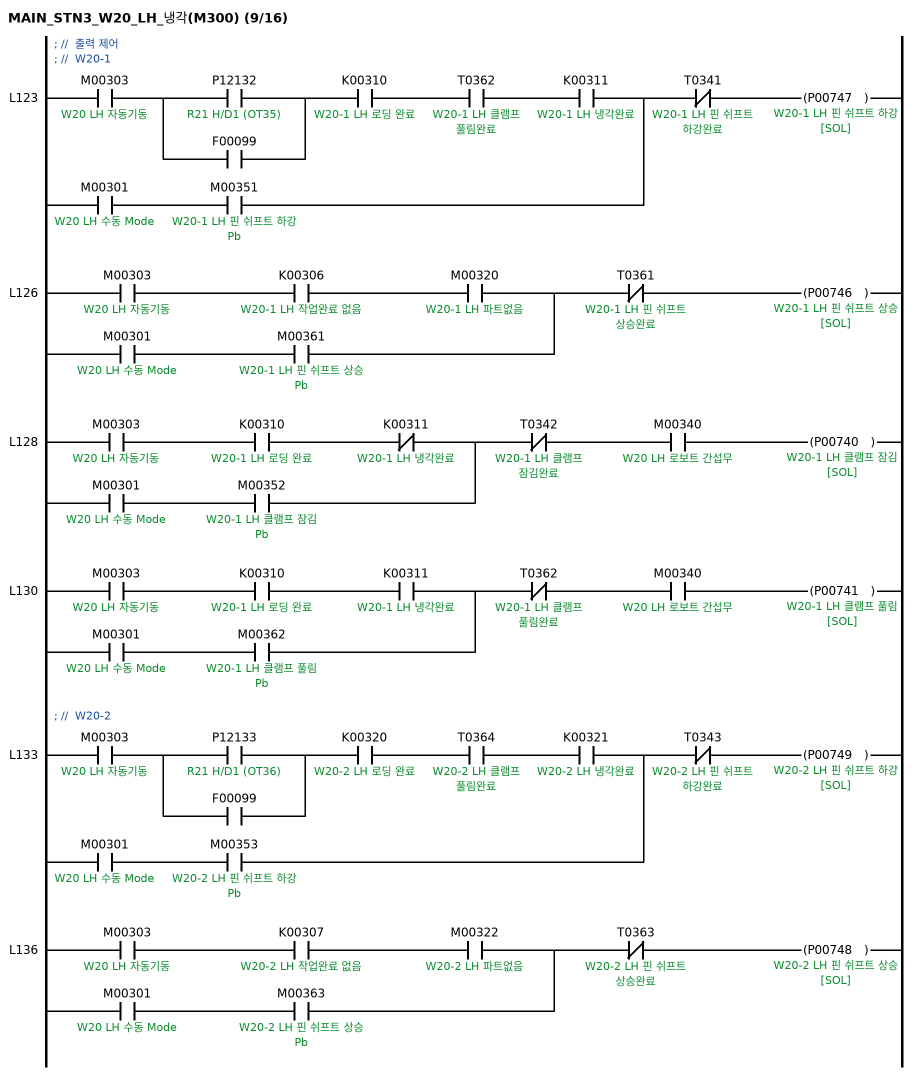
//     //  출력 제어
//     //  W20-1
; L123
LOAD      M00303	// W20 LH 자동기동
LOAD      P12132	// R21 H/D1 (OT35)
OR        F00099
AND LOAD
AND       K00310	// W20-1 LH 로딩 완료
AND       T0362	// W20-1 LH 클램프 풀림완료
AND       K00311	// W20-1 LH 냉각완료
LOAD      M00301	// W20 LH 수동 Mode
AND       M00351	// W20-1 LH 핀 쉬프트 하강 Pb
OR LOAD
AND NOT   T0341	// W20-1 LH 핀 쉬프트 하강완료
OUT       P00747	// W20-1 LH 핀 쉬프트 하강 [SOL]
; L126
LOAD      M00303	// W20 LH 자동기동
AND       K00306	// W20-1 LH 작업완료 없음
AND       M00320	// W20-1 LH 파트없음
LOAD      M00301	// W20 LH 수동 Mode
AND       M00361	// W20-1 LH 핀 쉬프트 상승 Pb
OR LOAD
AND NOT   T0361	// W20-1 LH 핀 쉬프트 상승완료
OUT       P00746	// W20-1 LH 핀 쉬프트 상승 [SOL]
; L128
LOAD      M00303	// W20 LH 자동기동
AND       K00310	// W20-1 LH 로딩 완료
AND NOT   K00311	// W20-1 LH 냉각완료
LOAD      M00301	// W20 LH 수동 Mode
AND       M00352	// W20-1 LH 클램프 잠김 Pb
OR LOAD
AND NOT   T0342	// W20-1 LH 클램프 잠김완료
AND       M00340	// W20 LH 로보트 간섭무
OUT       P00740	// W20-1 LH 클램프 잠김 [SOL]
; L130
LOAD      M00303	// W20 LH 자동기동
AND       K00310	// W20-1 LH 로딩 완료
AND       K00311	// W20-1 LH 냉각완료
LOAD      M00301	// W20 LH 수동 Mode
AND       M00362	// W20-1 LH 클램프 풀림 Pb
OR LOAD
AND NOT   T0362	// W20-1 LH 클램프 풀림완료
AND       M00340	// W20 LH 로보트 간섭무
OUT       P00741	// W20-1 LH 클램프 풀림 [SOL]
//     //  W20-2
; L133
LOAD      M00303	// W20 LH 자동기동
LOAD      P12133	// R21 H/D1 (OT36)
OR        F00099
AND LOAD
AND       K00320	// W20-2 LH 로딩 완료
AND       T0364	// W20-2 LH 클램프 풀림완료
AND       K00321	// W20-2 LH 냉각완료
LOAD      M00301	// W20 LH 수동 Mode
AND       M00353	// W20-2 LH 핀 쉬프트 하강 Pb
OR LOAD
AND NOT   T0343	// W20-2 LH 핀 쉬프트 하강완료
OUT       P00749	// W20-2 LH 핀 쉬프트 하강 [SOL]
; L136
LOAD      M00303	// W20 LH 자동기동
AND       K00307	// W20-2 LH 작업완료 없음
AND       M00322	// W20-2 LH 파트없음
LOAD      M00301	// W20 LH 수동 Mode
AND       M00363	// W20-2 LH 핀 쉬프트 상승 Pb
OR LOAD
AND NOT   T0363	// W20-2 LH 핀 쉬프트 상승완료
OUT       P00748	// W20-2 LH 핀 쉬프트 상승 [SOL]

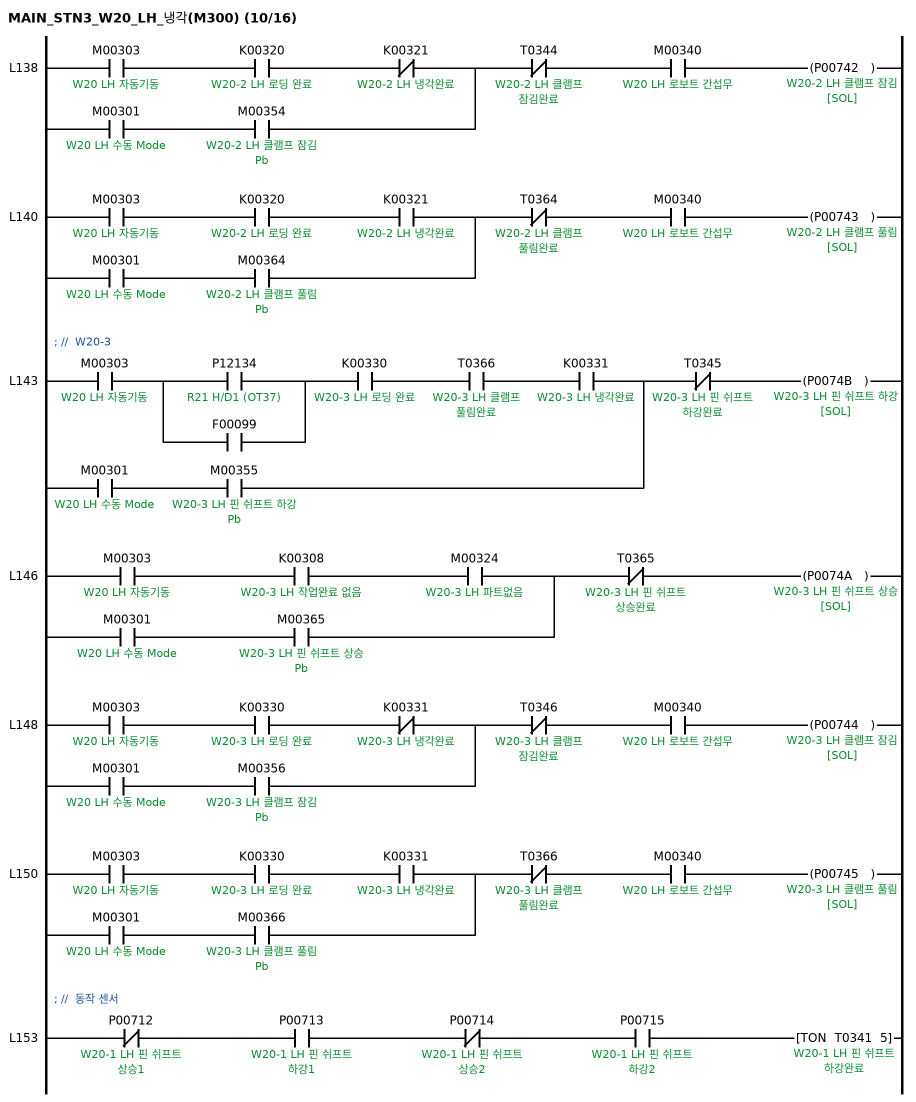
; L138
LOAD      M00303	// W20 LH 자동기동
AND       K00320	// W20-2 LH 로딩 완료
AND NOT   K00321	// W20-2 LH 냉각완료
LOAD      M00301	// W20 LH 수동 Mode
AND       M00354	// W20-2 LH 클램프 잠김 Pb
OR LOAD
AND NOT   T0344	// W20-2 LH 클램프 잠김완료
AND       M00340	// W20 LH 로보트 간섭무
OUT       P00742	// W20-2 LH 클램프 잠김 [SOL]
; L140
LOAD      M00303	// W20 LH 자동기동
AND       K00320	// W20-2 LH 로딩 완료
AND       K00321	// W20-2 LH 냉각완료
LOAD      M00301	// W20 LH 수동 Mode
AND       M00364	// W20-2 LH 클램프 풀림 Pb
OR LOAD
AND NOT   T0364	// W20-2 LH 클램프 풀림완료
AND       M00340	// W20 LH 로보트 간섭무
OUT       P00743	// W20-2 LH 클램프 풀림 [SOL]
//     //  W20-3
; L143
LOAD      M00303	// W20 LH 자동기동
LOAD      P12134	// R21 H/D1 (OT37)
OR        F00099
AND LOAD
AND       K00330	// W20-3 LH 로딩 완료
AND       T0366	// W20-3 LH 클램프 풀림완료
AND       K00331	// W20-3 LH 냉각완료
LOAD      M00301	// W20 LH 수동 Mode
AND       M00355	// W20-3 LH 핀 쉬프트 하강 Pb
OR LOAD
AND NOT   T0345	// W20-3 LH 핀 쉬프트 하강완료
OUT       P0074B	// W20-3 LH 핀 쉬프트 하강 [SOL]
; L146
LOAD      M00303	// W20 LH 자동기동
AND       K00308	// W20-3 LH 작업완료 없음
AND       M00324	// W20-3 LH 파트없음
LOAD      M00301	// W20 LH 수동 Mode
AND       M00365	// W20-3 LH 핀 쉬프트 상승 Pb
OR LOAD
AND NOT   T0365	// W20-3 LH 핀 쉬프트 상승완료
OUT       P0074A	// W20-3 LH 핀 쉬프트 상승 [SOL]
; L148
LOAD      M00303	// W20 LH 자동기동
AND       K00330	// W20-3 LH 로딩 완료
AND NOT   K00331	// W20-3 LH 냉각완료
LOAD      M00301	// W20 LH 수동 Mode
AND       M00356	// W20-3 LH 클램프 잠김 Pb
OR LOAD
AND NOT   T0346	// W20-3 LH 클램프 잠김완료
AND       M00340	// W20 LH 로보트 간섭무
OUT       P00744	// W20-3 LH 클램프 잠김 [SOL]
; L150
LOAD      M00303	// W20 LH 자동기동
AND       K00330	// W20-3 LH 로딩 완료
AND       K00331	// W20-3 LH 냉각완료
LOAD      M00301	// W20 LH 수동 Mode
AND       M00366	// W20-3 LH 클램프 풀림 Pb
OR LOAD
AND NOT   T0366	// W20-3 LH 클램프 풀림완료
AND       M00340	// W20 LH 로보트 간섭무
OUT       P00745	// W20-3 LH 클램프 풀림 [SOL]
//   //  동작 센서
; L153
LOAD NOT  P00712	// W20-1 LH 핀 쉬프트 상승1
AND       P00713	// W20-1 LH 핀 쉬프트 하강1
AND NOT   P00714	// W20-1 LH 핀 쉬프트 상승2
AND       P00715	// W20-1 LH 핀 쉬프트 하강2
TON       T0341 5	// W20-1 LH 핀 쉬프트 하강완료

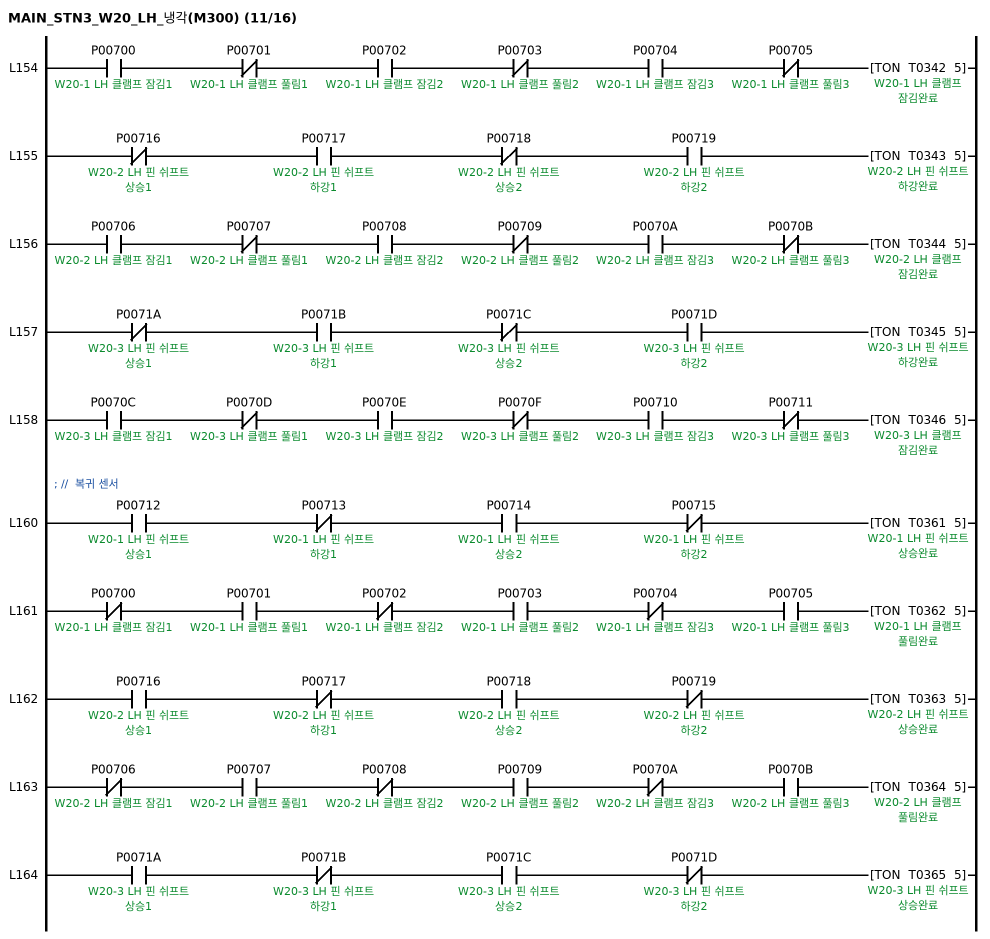
; L154
LOAD      P00700	// W20-1 LH 클램프 잠김1
AND NOT   P00701	// W20-1 LH 클램프 풀림1
AND       P00702	// W20-1 LH 클램프 잠김2
AND NOT   P00703	// W20-1 LH 클램프 풀림2
AND       P00704	// W20-1 LH 클램프 잠김3
AND NOT   P00705	// W20-1 LH 클램프 풀림3
TON       T0342 5	// W20-1 LH 클램프 잠김완료
; L155
LOAD NOT  P00716	// W20-2 LH 핀 쉬프트 상승1
AND       P00717	// W20-2 LH 핀 쉬프트 하강1
AND NOT   P00718	// W20-2 LH 핀 쉬프트 상승2
AND       P00719	// W20-2 LH 핀 쉬프트 하강2
TON       T0343 5	// W20-2 LH 핀 쉬프트 하강완료
; L156
LOAD      P00706	// W20-2 LH 클램프 잠김1
AND NOT   P00707	// W20-2 LH 클램프 풀림1
AND       P00708	// W20-2 LH 클램프 잠김2
AND NOT   P00709	// W20-2 LH 클램프 풀림2
AND       P0070A	// W20-2 LH 클램프 잠김3
AND NOT   P0070B	// W20-2 LH 클램프 풀림3
TON       T0344 5	// W20-2 LH 클램프 잠김완료
; L157
LOAD NOT  P0071A	// W20-3 LH 핀 쉬프트 상승1
AND       P0071B	// W20-3 LH 핀 쉬프트 하강1
AND NOT   P0071C	// W20-3 LH 핀 쉬프트 상승2
AND       P0071D	// W20-3 LH 핀 쉬프트 하강2
TON       T0345 5	// W20-3 LH 핀 쉬프트 하강완료
; L158
LOAD      P0070C	// W20-3 LH 클램프 잠김1
AND NOT   P0070D	// W20-3 LH 클램프 풀림1
AND       P0070E	// W20-3 LH 클램프 잠김2
AND NOT   P0070F	// W20-3 LH 클램프 풀림2
AND       P00710	// W20-3 LH 클램프 잠김3
AND NOT   P00711	// W20-3 LH 클램프 풀림3
TON       T0346 5	// W20-3 LH 클램프 잠김완료
//   //  복귀 센서
; L160
LOAD      P00712	// W20-1 LH 핀 쉬프트 상승1
AND NOT   P00713	// W20-1 LH 핀 쉬프트 하강1
AND       P00714	// W20-1 LH 핀 쉬프트 상승2
AND NOT   P00715	// W20-1 LH 핀 쉬프트 하강2
TON       T0361 5	// W20-1 LH 핀 쉬프트 상승완료
; L161
LOAD NOT  P00700	// W20-1 LH 클램프 잠김1
AND       P00701	// W20-1 LH 클램프 풀림1
AND NOT   P00702	// W20-1 LH 클램프 잠김2
AND       P00703	// W20-1 LH 클램프 풀림2
AND NOT   P00704	// W20-1 LH 클램프 잠김3
AND       P00705	// W20-1 LH 클램프 풀림3
TON       T0362 5	// W20-1 LH 클램프 풀림완료
; L162
LOAD      P00716	// W20-2 LH 핀 쉬프트 상승1
AND NOT   P00717	// W20-2 LH 핀 쉬프트 하강1
AND       P00718	// W20-2 LH 핀 쉬프트 상승2
AND NOT   P00719	// W20-2 LH 핀 쉬프트 하강2
TON       T0363 5	// W20-2 LH 핀 쉬프트 상승완료
; L163
LOAD NOT  P00706	// W20-2 LH 클램프 잠김1
AND       P00707	// W20-2 LH 클램프 풀림1
AND NOT   P00708	// W20-2 LH 클램프 잠김2
AND       P00709	// W20-2 LH 클램프 풀림2
AND NOT   P0070A	// W20-2 LH 클램프 잠김3
AND       P0070B	// W20-2 LH 클램프 풀림3
TON       T0364 5	// W20-2 LH 클램프 풀림완료
; L164
LOAD      P0071A	// W20-3 LH 핀 쉬프트 상승1
AND NOT   P0071B	// W20-3 LH 핀 쉬프트 하강1
AND       P0071C	// W20-3 LH 핀 쉬프트 상승2
AND NOT   P0071D	// W20-3 LH 핀 쉬프트 하강2
TON       T0365 5	// W20-3 LH 핀 쉬프트 상승완료

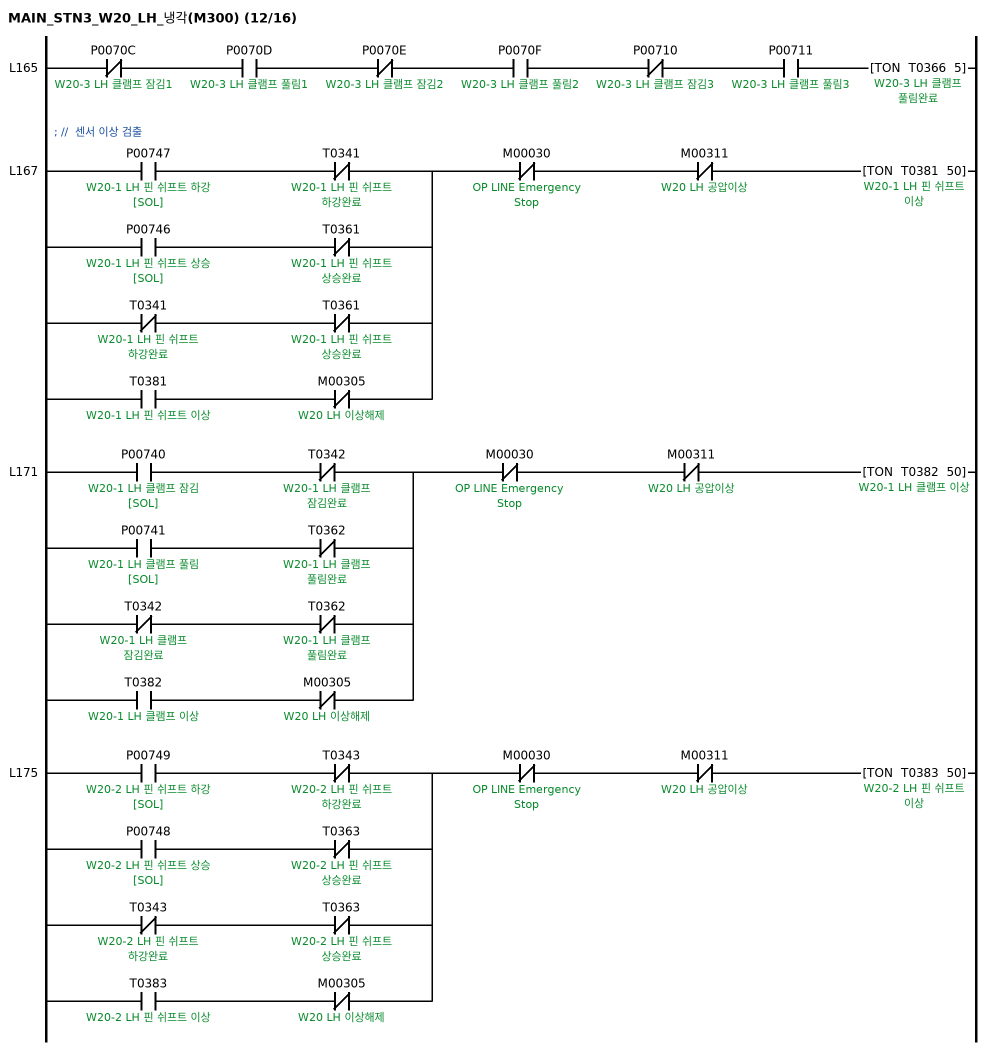
; L165
LOAD NOT  P0070C	// W20-3 LH 클램프 잠김1
AND       P0070D	// W20-3 LH 클램프 풀림1
AND NOT   P0070E	// W20-3 LH 클램프 잠김2
AND       P0070F	// W20-3 LH 클램프 풀림2
AND NOT   P00710	// W20-3 LH 클램프 잠김3
AND       P00711	// W20-3 LH 클램프 풀림3
TON       T0366 5	// W20-3 LH 클램프 풀림완료
//     //  센서 이상 검출
; L167
LOAD      P00747	// W20-1 LH 핀 쉬프트 하강 [SOL]
AND NOT   T0341	// W20-1 LH 핀 쉬프트 하강완료
LOAD      P00746	// W20-1 LH 핀 쉬프트 상승 [SOL]
AND NOT   T0361	// W20-1 LH 핀 쉬프트 상승완료
OR LOAD
LOAD NOT  T0341	// W20-1 LH 핀 쉬프트 하강완료
AND NOT   T0361	// W20-1 LH 핀 쉬프트 상승완료
OR LOAD
LOAD      T0381	// W20-1 LH 핀 쉬프트 이상
AND NOT   M00305	// W20 LH 이상해제
OR LOAD
AND NOT   M00030	// OP LINE Emergency Stop
AND NOT   M00311	// W20 LH 공압이상
TON       T0381 50	// W20-1 LH 핀 쉬프트 이상
; L171
LOAD      P00740	// W20-1 LH 클램프 잠김 [SOL]
AND NOT   T0342	// W20-1 LH 클램프 잠김완료
LOAD      P00741	// W20-1 LH 클램프 풀림 [SOL]
AND NOT   T0362	// W20-1 LH 클램프 풀림완료
OR LOAD
LOAD NOT  T0342	// W20-1 LH 클램프 잠김완료
AND NOT   T0362	// W20-1 LH 클램프 풀림완료
OR LOAD
LOAD      T0382	// W20-1 LH 클램프 이상
AND NOT   M00305	// W20 LH 이상해제
OR LOAD
AND NOT   M00030	// OP LINE Emergency Stop
AND NOT   M00311	// W20 LH 공압이상
TON       T0382 50	// W20-1 LH 클램프 이상
; L175
LOAD      P00749	// W20-2 LH 핀 쉬프트 하강 [SOL]
AND NOT   T0343	// W20-2 LH 핀 쉬프트 하강완료
LOAD      P00748	// W20-2 LH 핀 쉬프트 상승 [SOL]
AND NOT   T0363	// W20-2 LH 핀 쉬프트 상승완료
OR LOAD
LOAD NOT  T0343	// W20-2 LH 핀 쉬프트 하강완료
AND NOT   T0363	// W20-2 LH 핀 쉬프트 상승완료
OR LOAD
LOAD      T0383	// W20-2 LH 핀 쉬프트 이상
AND NOT   M00305	// W20 LH 이상해제
OR LOAD
AND NOT   M00030	// OP LINE Emergency Stop
AND NOT   M00311	// W20 LH 공압이상
TON       T0383 50	// W20-2 LH 핀 쉬프트 이상

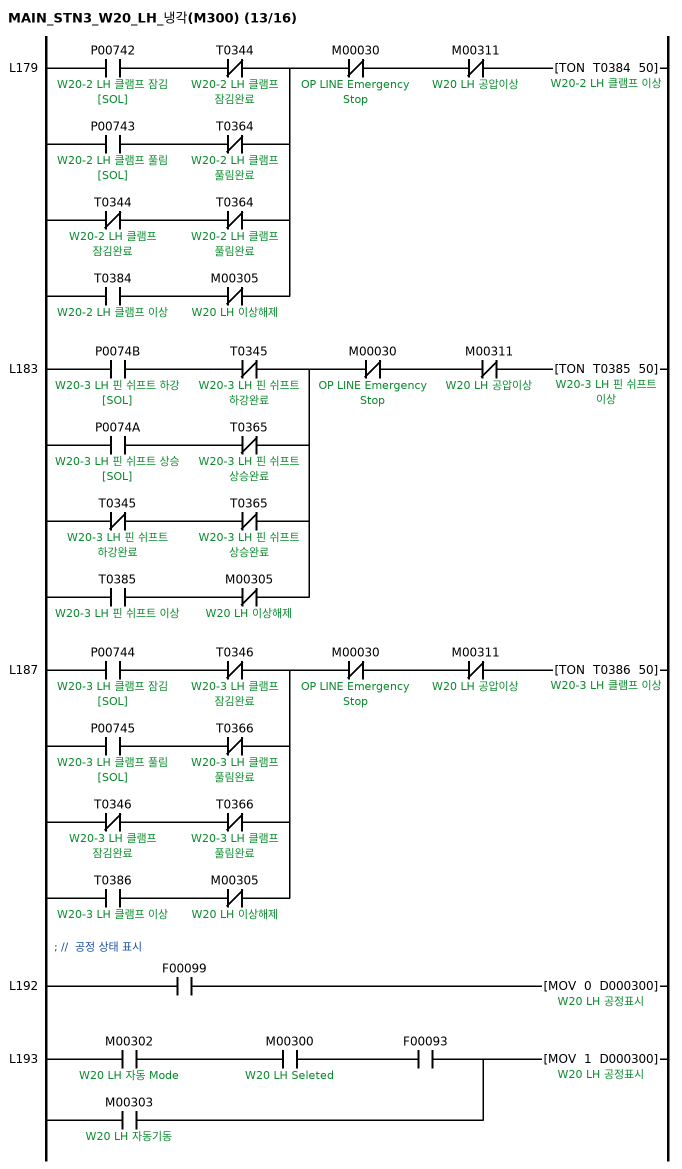
; L179
LOAD      P00742	// W20-2 LH 클램프 잠김 [SOL]
AND NOT   T0344	// W20-2 LH 클램프 잠김완료
LOAD      P00743	// W20-2 LH 클램프 풀림 [SOL]
AND NOT   T0364	// W20-2 LH 클램프 풀림완료
OR LOAD
LOAD NOT  T0344	// W20-2 LH 클램프 잠김완료
AND NOT   T0364	// W20-2 LH 클램프 풀림완료
OR LOAD
LOAD      T0384	// W20-2 LH 클램프 이상
AND NOT   M00305	// W20 LH 이상해제
OR LOAD
AND NOT   M00030	// OP LINE Emergency Stop
AND NOT   M00311	// W20 LH 공압이상
TON       T0384 50	// W20-2 LH 클램프 이상
; L183
LOAD      P0074B	// W20-3 LH 핀 쉬프트 하강 [SOL]
AND NOT   T0345	// W20-3 LH 핀 쉬프트 하강완료
LOAD      P0074A	// W20-3 LH 핀 쉬프트 상승 [SOL]
AND NOT   T0365	// W20-3 LH 핀 쉬프트 상승완료
OR LOAD
LOAD NOT  T0345	// W20-3 LH 핀 쉬프트 하강완료
AND NOT   T0365	// W20-3 LH 핀 쉬프트 상승완료
OR LOAD
LOAD      T0385	// W20-3 LH 핀 쉬프트 이상
AND NOT   M00305	// W20 LH 이상해제
OR LOAD
AND NOT   M00030	// OP LINE Emergency Stop
AND NOT   M00311	// W20 LH 공압이상
TON       T0385 50	// W20-3 LH 핀 쉬프트 이상
; L187
LOAD      P00744	// W20-3 LH 클램프 잠김 [SOL]
AND NOT   T0346	// W20-3 LH 클램프 잠김완료
LOAD      P00745	// W20-3 LH 클램프 풀림 [SOL]
AND NOT   T0366	// W20-3 LH 클램프 풀림완료
OR LOAD
LOAD NOT  T0346	// W20-3 LH 클램프 잠김완료
AND NOT   T0366	// W20-3 LH 클램프 풀림완료
OR LOAD
LOAD      T0386	// W20-3 LH 클램프 이상
AND NOT   M00305	// W20 LH 이상해제
OR LOAD
AND NOT   M00030	// OP LINE Emergency Stop
AND NOT   M00311	// W20 LH 공압이상
TON       T0386 50	// W20-3 LH 클램프 이상
//   //  공정 상태 표시
; L192
LOAD      F00099
MOV       0 D000300	// W20 LH 공정표시
; L193
LOAD      M00302	// W20 LH 자동 Mode
AND       M00300	// W20 LH Seleted
AND       F00093
OR        M00303	// W20 LH 자동기동
MOV       1 D000300	// W20 LH 공정표시

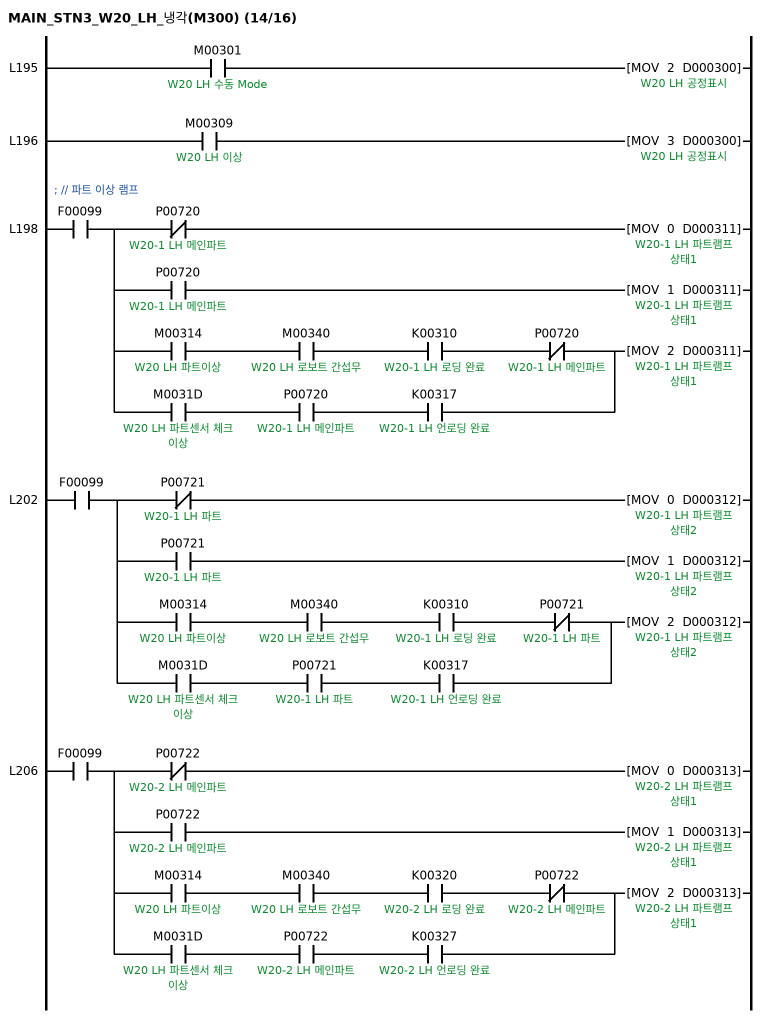
; L195
LOAD      M00301	// W20 LH 수동 Mode
MOV       2 D000300	// W20 LH 공정표시
; L196
LOAD      M00309	// W20 LH 이상
MOV       3 D000300	// W20 LH 공정표시
//   // 파트 이상 램프
; L198
LOAD      F00099
MPUSH
AND NOT   P00720	// W20-1 LH 메인파트
MOV       0 D000311	// W20-1 LH 파트램프 상태1
MLOAD
AND       P00720	// W20-1 LH 메인파트
MOV       1 D000311	// W20-1 LH 파트램프 상태1
MPOP
LOAD      M00314	// W20 LH 파트이상
AND       M00340	// W20 LH 로보트 간섭무
AND       K00310	// W20-1 LH 로딩 완료
AND NOT   P00720	// W20-1 LH 메인파트
LOAD      M0031D	// W20 LH 파트센서 체크 이상
AND       P00720	// W20-1 LH 메인파트
AND       K00317	// W20-1 LH 언로딩 완료
OR LOAD
AND LOAD
MOV       2 D000311	// W20-1 LH 파트램프 상태1
; L202
LOAD      F00099
MPUSH
AND NOT   P00721	// W20-1 LH 파트
MOV       0 D000312	// W20-1 LH 파트램프 상태2
MLOAD
AND       P00721	// W20-1 LH 파트
MOV       1 D000312	// W20-1 LH 파트램프 상태2
MPOP
LOAD      M00314	// W20 LH 파트이상
AND       M00340	// W20 LH 로보트 간섭무
AND       K00310	// W20-1 LH 로딩 완료
AND NOT   P00721	// W20-1 LH 파트
LOAD      M0031D	// W20 LH 파트센서 체크 이상
AND       P00721	// W20-1 LH 파트
AND       K00317	// W20-1 LH 언로딩 완료
OR LOAD
AND LOAD
MOV       2 D000312	// W20-1 LH 파트램프 상태2
; L206
LOAD      F00099
MPUSH
AND NOT   P00722	// W20-2 LH 메인파트
MOV       0 D000313	// W20-2 LH 파트램프 상태1
MLOAD
AND       P00722	// W20-2 LH 메인파트
MOV       1 D000313	// W20-2 LH 파트램프 상태1
MPOP
LOAD      M00314	// W20 LH 파트이상
AND       M00340	// W20 LH 로보트 간섭무
AND       K00320	// W20-2 LH 로딩 완료
AND NOT   P00722	// W20-2 LH 메인파트
LOAD      M0031D	// W20 LH 파트센서 체크 이상
AND       P00722	// W20-2 LH 메인파트
AND       K00327	// W20-2 LH 언로딩 완료
OR LOAD
AND LOAD
MOV       2 D000313	// W20-2 LH 파트램프 상태1

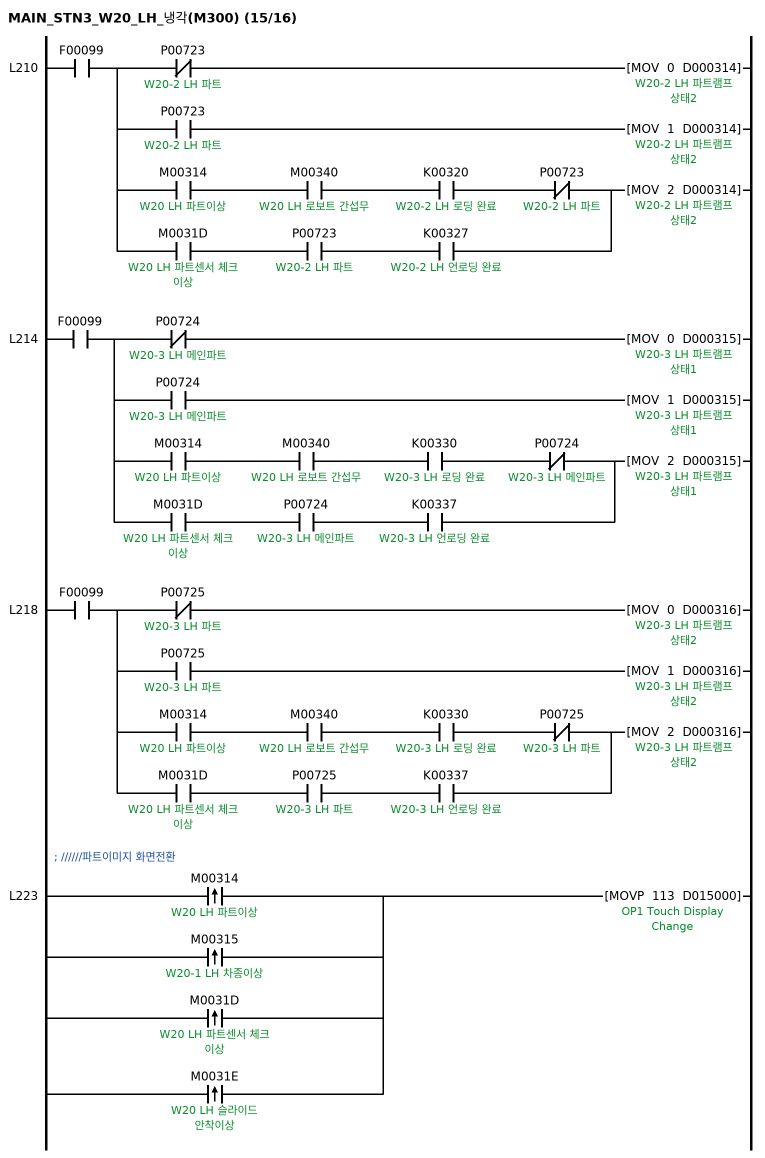
; L210
LOAD      F00099
MPUSH
AND NOT   P00723	// W20-2 LH 파트
MOV       0 D000314	// W20-2 LH 파트램프 상태2
MLOAD
AND       P00723	// W20-2 LH 파트
MOV       1 D000314	// W20-2 LH 파트램프 상태2
MPOP
LOAD      M00314	// W20 LH 파트이상
AND       M00340	// W20 LH 로보트 간섭무
AND       K00320	// W20-2 LH 로딩 완료
AND NOT   P00723	// W20-2 LH 파트
LOAD      M0031D	// W20 LH 파트센서 체크 이상
AND       P00723	// W20-2 LH 파트
AND       K00327	// W20-2 LH 언로딩 완료
OR LOAD
AND LOAD
MOV       2 D000314	// W20-2 LH 파트램프 상태2
; L214
LOAD      F00099
MPUSH
AND NOT   P00724	// W20-3 LH 메인파트
MOV       0 D000315	// W20-3 LH 파트램프 상태1
MLOAD
AND       P00724	// W20-3 LH 메인파트
MOV       1 D000315	// W20-3 LH 파트램프 상태1
MPOP
LOAD      M00314	// W20 LH 파트이상
AND       M00340	// W20 LH 로보트 간섭무
AND       K00330	// W20-3 LH 로딩 완료
AND NOT   P00724	// W20-3 LH 메인파트
LOAD      M0031D	// W20 LH 파트센서 체크 이상
AND       P00724	// W20-3 LH 메인파트
AND       K00337	// W20-3 LH 언로딩 완료
OR LOAD
AND LOAD
MOV       2 D000315	// W20-3 LH 파트램프 상태1
; L218
LOAD      F00099
MPUSH
AND NOT   P00725	// W20-3 LH 파트
MOV       0 D000316	// W20-3 LH 파트램프 상태2
MLOAD
AND       P00725	// W20-3 LH 파트
MOV       1 D000316	// W20-3 LH 파트램프 상태2
MPOP
LOAD      M00314	// W20 LH 파트이상
AND       M00340	// W20 LH 로보트 간섭무
AND       K00330	// W20-3 LH 로딩 완료
AND NOT   P00725	// W20-3 LH 파트
LOAD      M0031D	// W20 LH 파트센서 체크 이상
AND       P00725	// W20-3 LH 파트
AND       K00337	// W20-3 LH 언로딩 완료
OR LOAD
AND LOAD
MOV       2 D000316	// W20-3 LH 파트램프 상태2
// //////파트이미지 화면전환
; L223
LOADP     M00314	// W20 LH 파트이상
ORP       M00315	// W20-1 LH 차종이상
ORP       M0031D	// W20 LH 파트센서 체크 이상
ORP       M0031E	// W20 LH 슬라이드 안착이상
MOVP      113 D015000	// OP1 Touch Display Change

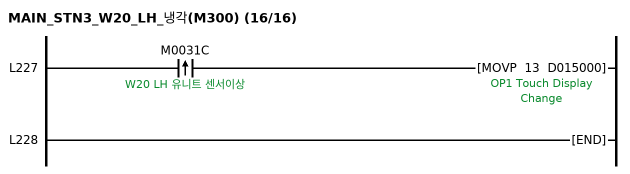
; L227
LOADP     M0031C	// W20 LH 유니트 센서이상
MOVP      13 D015000	// OP1 Touch Display Change
; L228
END

PROGRAM MAIN_STN4_W20_RH_냉각(M400) (task: 스캔 프로그램)

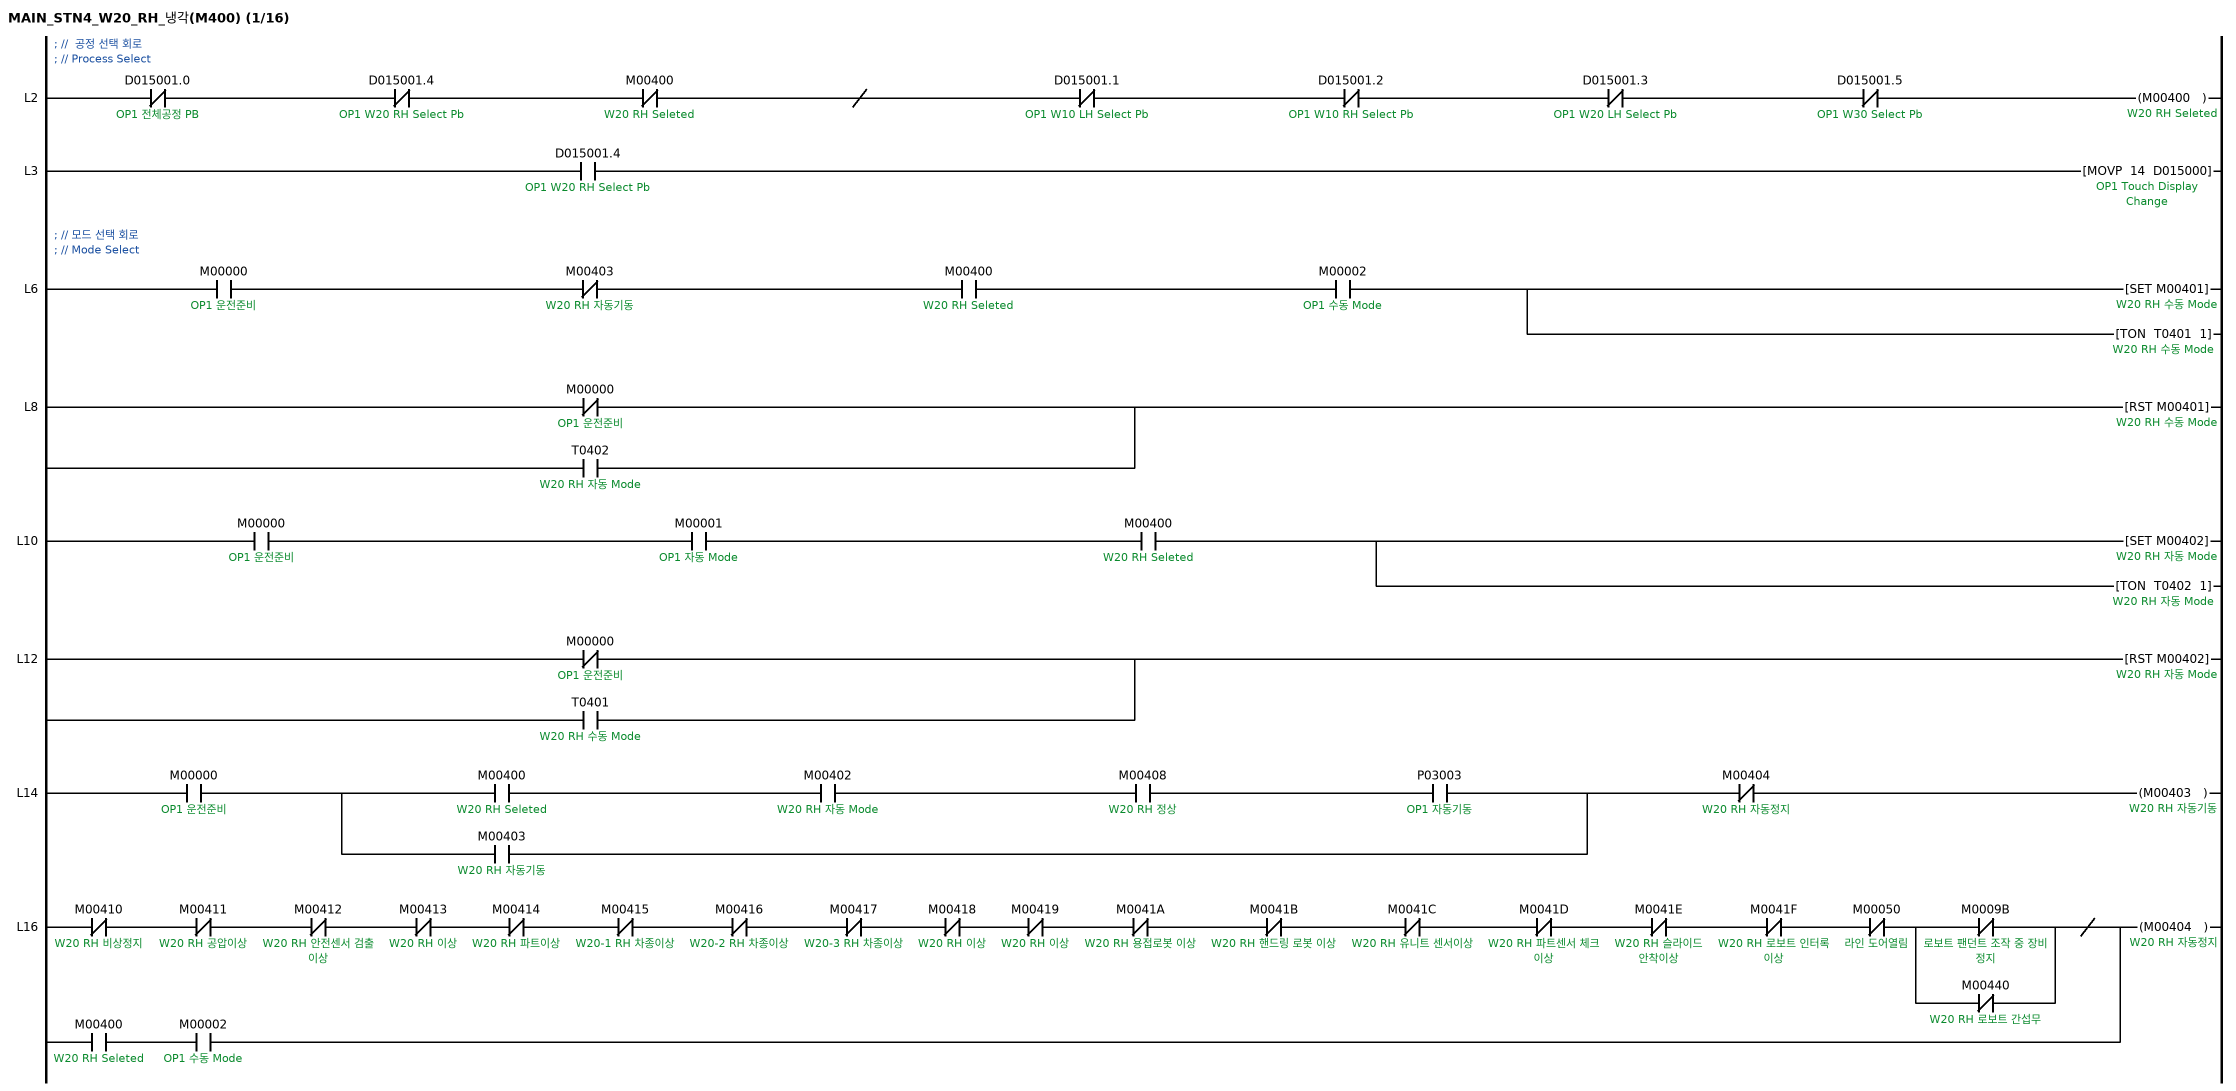
//   //  공정 선택 회로
//   // Process Select
; L2
LOAD NOT  D015001.0	// OP1 전체공정 PB
AND NOT   D015001.4	// OP1 W20 RH Select Pb
AND NOT   M00400	// W20 RH Seleted
NOT
AND NOT   D015001.1	// OP1 W10 LH Select Pb
AND NOT   D015001.2	// OP1 W10 RH Select Pb
AND NOT   D015001.3	// OP1 W20 LH Select Pb
AND NOT   D015001.5	// OP1 W30 Select Pb
OUT       M00400	// W20 RH Seleted
; L3
LOAD      D015001.4	// OP1 W20 RH Select Pb
MOVP      14 D015000	// OP1 Touch Display Change
// // 모드 선택 회로
//   // Mode Select
; L6
LOAD      M00000	// OP1 운전준비
AND NOT   M00403	// W20 RH 자동기동
AND       M00400	// W20 RH Seleted
AND       M00002	// OP1 수동 Mode
SET       M00401	// W20 RH 수동 Mode
TON       T0401 1	// W20 RH 수동 Mode
; L8
LOAD NOT  M00000	// OP1 운전준비
OR        T0402	// W20 RH 자동 Mode
RST       M00401	// W20 RH 수동 Mode
; L10
LOAD      M00000	// OP1 운전준비
AND       M00001	// OP1 자동 Mode
AND       M00400	// W20 RH Seleted
SET       M00402	// W20 RH 자동 Mode
TON       T0402 1	// W20 RH 자동 Mode
; L12
LOAD NOT  M00000	// OP1 운전준비
OR        T0401	// W20 RH 수동 Mode
RST       M00402	// W20 RH 자동 Mode
; L14
LOAD      M00000	// OP1 운전준비
LOAD      M00400	// W20 RH Seleted
AND       M00402	// W20 RH 자동 Mode
AND       M00408	// W20 RH 정상
AND       P03003	// OP1 자동기동
OR        M00403	// W20 RH 자동기동
AND LOAD
AND NOT   M00404	// W20 RH 자동정지
OUT       M00403	// W20 RH 자동기동
; L16
LOAD NOT  M00410	// W20 RH 비상정지
AND NOT   M00411	// W20 RH 공압이상
AND NOT   M00412	// W20 RH 안전센서 검출 이상
AND NOT   M00413	// W20 RH 이상
AND NOT   M00414	// W20 RH 파트이상
AND NOT   M00415	// W20-1 RH 차종이상
AND NOT   M00416	// W20-2 RH 차종이상
AND NOT   M00417	// W20-3 RH 차종이상
AND NOT   M00418	// W20 RH 이상
AND NOT   M00419	// W20 RH 이상
AND NOT   M0041A	// W20 RH 용접로봇 이상
AND NOT   M0041B	// W20 RH 핸드링 로봇 이상
AND NOT   M0041C	// W20 RH 유니트 센서이상
AND NOT   M0041D	// W20 RH 파트센서 체크 이상
AND NOT   M0041E	// W20 RH 슬라이드 안착이상
AND NOT   M0041F	// W20 RH 로보트 인터록 이상
AND NOT   M00050	// 라인 도어열림
LOAD NOT  M0009B	// 로보트 팬던트 조작 중 장비 정지
OR NOT    M00440	// W20 RH 로보트 간섭무
AND LOAD
NOT
LOAD      M00400	// W20 RH Seleted
AND       M00002	// OP1 수동 Mode
OR LOAD
OUT       M00404	// W20 RH 자동정지

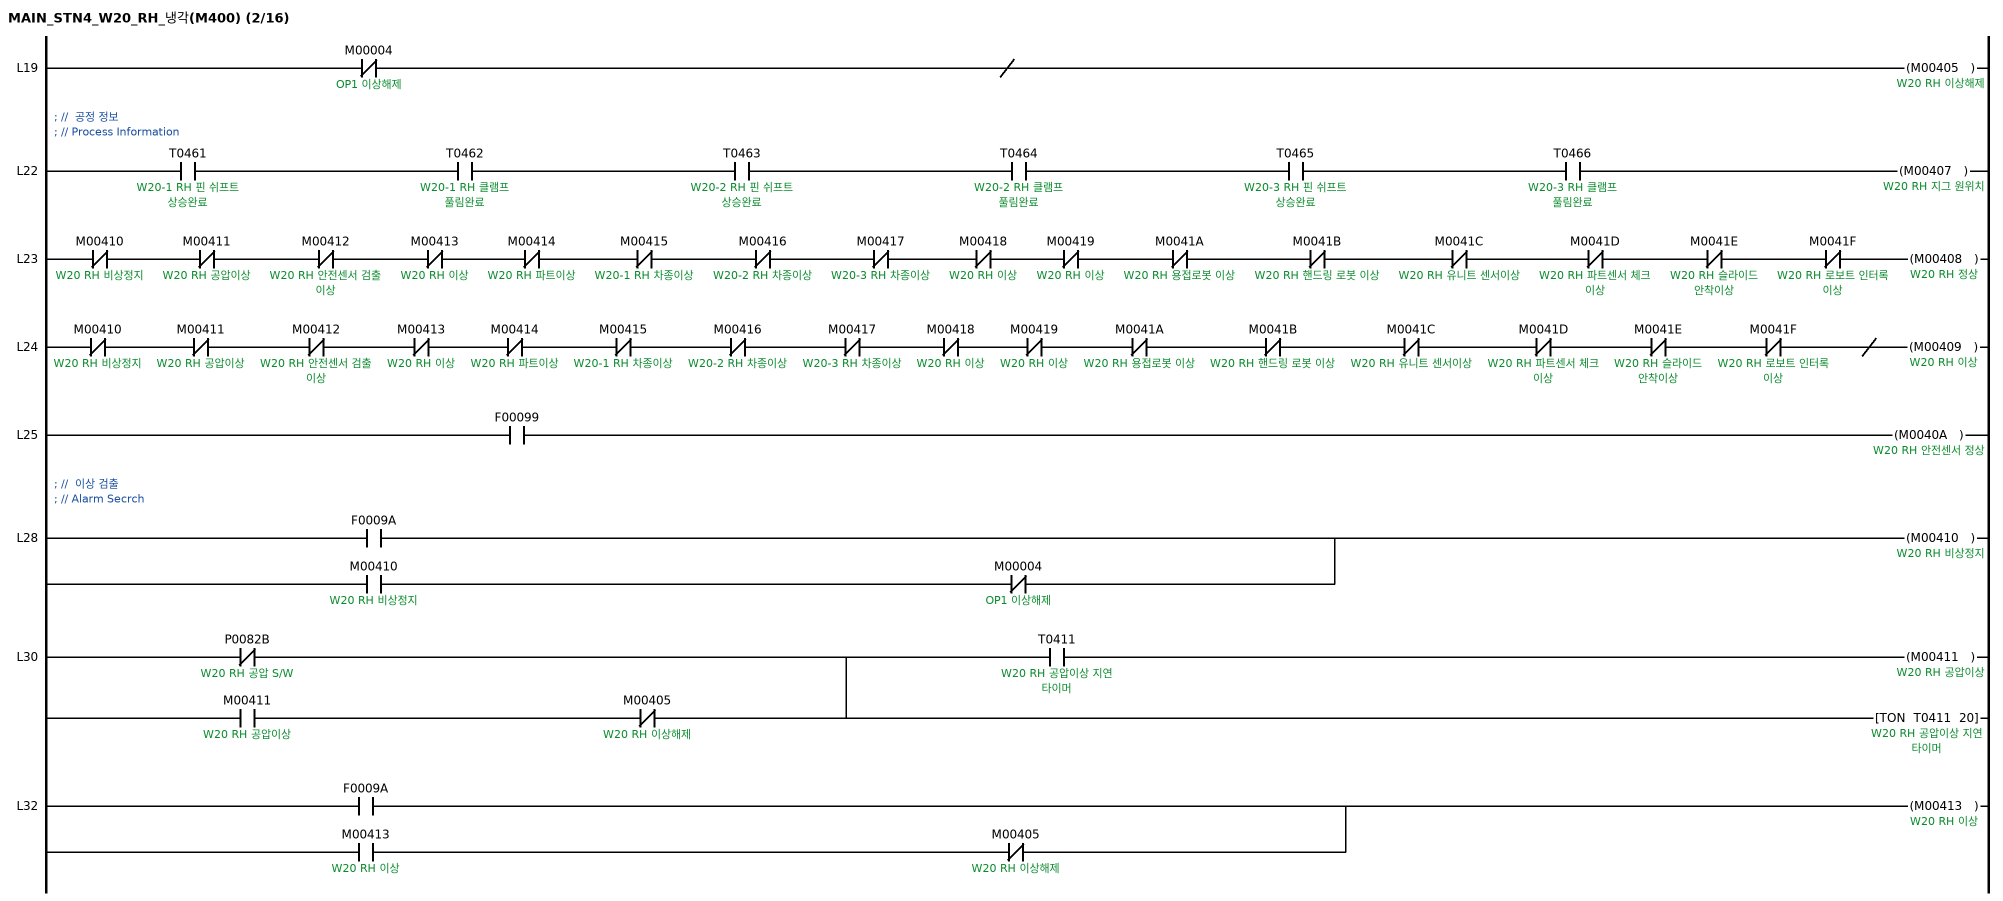
; L19
LOAD NOT  M00004	// OP1 이상해제
NOT
OUT       M00405	// W20 RH 이상해제
//   //  공정 정보
//   // Process Information
; L22
LOAD      T0461	// W20-1 RH 핀 쉬프트 상승완료
AND       T0462	// W20-1 RH 클램프 풀림완료
AND       T0463	// W20-2 RH 핀 쉬프트 상승완료
AND       T0464	// W20-2 RH 클램프 풀림완료
AND       T0465	// W20-3 RH 핀 쉬프트 상승완료
AND       T0466	// W20-3 RH 클램프 풀림완료
OUT       M00407	// W20 RH 지그 원위치
; L23
LOAD NOT  M00410	// W20 RH 비상정지
AND NOT   M00411	// W20 RH 공압이상
AND NOT   M00412	// W20 RH 안전센서 검출 이상
AND NOT   M00413	// W20 RH 이상
AND NOT   M00414	// W20 RH 파트이상
AND NOT   M00415	// W20-1 RH 차종이상
AND NOT   M00416	// W20-2 RH 차종이상
AND NOT   M00417	// W20-3 RH 차종이상
AND NOT   M00418	// W20 RH 이상
AND NOT   M00419	// W20 RH 이상
AND NOT   M0041A	// W20 RH 용접로봇 이상
AND NOT   M0041B	// W20 RH 핸드링 로봇 이상
AND NOT   M0041C	// W20 RH 유니트 센서이상
AND NOT   M0041D	// W20 RH 파트센서 체크 이상
AND NOT   M0041E	// W20 RH 슬라이드 안착이상
AND NOT   M0041F	// W20 RH 로보트 인터록 이상
OUT       M00408	// W20 RH 정상
; L24
LOAD NOT  M00410	// W20 RH 비상정지
AND NOT   M00411	// W20 RH 공압이상
AND NOT   M00412	// W20 RH 안전센서 검출 이상
AND NOT   M00413	// W20 RH 이상
AND NOT   M00414	// W20 RH 파트이상
AND NOT   M00415	// W20-1 RH 차종이상
AND NOT   M00416	// W20-2 RH 차종이상
AND NOT   M00417	// W20-3 RH 차종이상
AND NOT   M00418	// W20 RH 이상
AND NOT   M00419	// W20 RH 이상
AND NOT   M0041A	// W20 RH 용접로봇 이상
AND NOT   M0041B	// W20 RH 핸드링 로봇 이상
AND NOT   M0041C	// W20 RH 유니트 센서이상
AND NOT   M0041D	// W20 RH 파트센서 체크 이상
AND NOT   M0041E	// W20 RH 슬라이드 안착이상
AND NOT   M0041F	// W20 RH 로보트 인터록 이상
NOT
OUT       M00409	// W20 RH 이상
; L25
LOAD      F00099
OUT       M0040A	// W20 RH 안전센서 정상
//   //  이상 검출
//   // Alarm Secrch
; L28
LOAD      F0009A
LOAD      M00410	// W20 RH 비상정지
AND NOT   M00004	// OP1 이상해제
OR LOAD
OUT       M00410	// W20 RH 비상정지
; L30
LOAD NOT  P0082B	// W20 RH 공압 S/W
LOAD      M00411	// W20 RH 공압이상
AND NOT   M00405	// W20 RH 이상해제
OR LOAD
MPUSH
AND       T0411	// W20 RH 공압이상 지연 타이머
OUT       M00411	// W20 RH 공압이상
MPOP
TON       T0411 20	// W20 RH 공압이상 지연 타이머
; L32
LOAD      F0009A
LOAD      M00413	// W20 RH 이상
AND NOT   M00405	// W20 RH 이상해제
OR LOAD
OUT       M00413	// W20 RH 이상

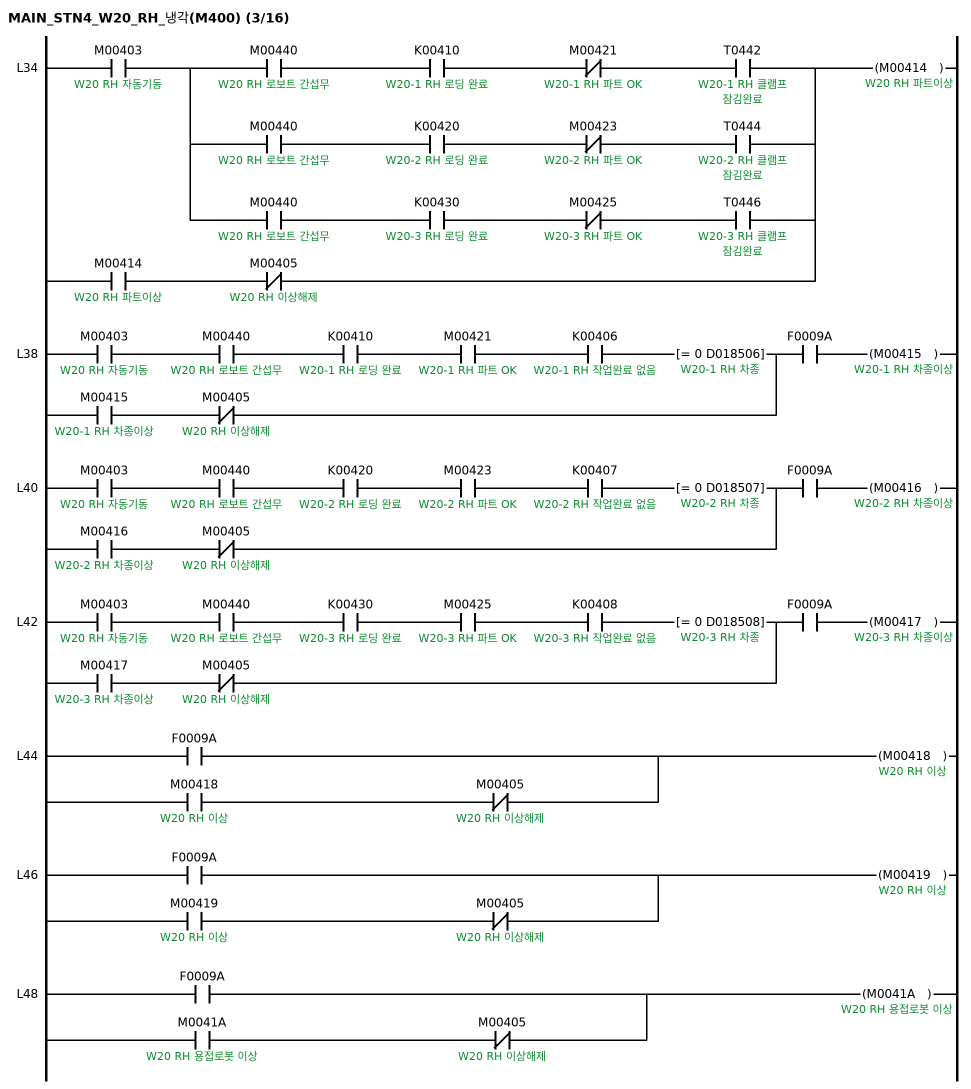
; L34
LOAD      M00403	// W20 RH 자동기동
LOAD      M00440	// W20 RH 로보트 간섭무
AND       K00410	// W20-1 RH 로딩 완료
AND NOT   M00421	// W20-1 RH 파트 OK
AND       T0442	// W20-1 RH 클램프 잠김완료
LOAD      M00440	// W20 RH 로보트 간섭무
AND       K00420	// W20-2 RH 로딩 완료
AND NOT   M00423	// W20-2 RH 파트 OK
AND       T0444	// W20-2 RH 클램프 잠김완료
OR LOAD
LOAD      M00440	// W20 RH 로보트 간섭무
AND       K00430	// W20-3 RH 로딩 완료
AND NOT   M00425	// W20-3 RH 파트 OK
AND       T0446	// W20-3 RH 클램프 잠김완료
OR LOAD
AND LOAD
LOAD      M00414	// W20 RH 파트이상
AND NOT   M00405	// W20 RH 이상해제
OR LOAD
OUT       M00414	// W20 RH 파트이상
; L38
LOAD      M00403	// W20 RH 자동기동
AND       M00440	// W20 RH 로보트 간섭무
AND       K00410	// W20-1 RH 로딩 완료
AND       M00421	// W20-1 RH 파트 OK
AND       K00406	// W20-1 RH 작업완료 없음
AND=      0 D018506	// W20-1 RH 차종
LOAD      M00415	// W20-1 RH 차종이상
AND NOT   M00405	// W20 RH 이상해제
OR LOAD
AND       F0009A
OUT       M00415	// W20-1 RH 차종이상
; L40
LOAD      M00403	// W20 RH 자동기동
AND       M00440	// W20 RH 로보트 간섭무
AND       K00420	// W20-2 RH 로딩 완료
AND       M00423	// W20-2 RH 파트 OK
AND       K00407	// W20-2 RH 작업완료 없음
AND=      0 D018507	// W20-2 RH 차종
LOAD      M00416	// W20-2 RH 차종이상
AND NOT   M00405	// W20 RH 이상해제
OR LOAD
AND       F0009A
OUT       M00416	// W20-2 RH 차종이상
; L42
LOAD      M00403	// W20 RH 자동기동
AND       M00440	// W20 RH 로보트 간섭무
AND       K00430	// W20-3 RH 로딩 완료
AND       M00425	// W20-3 RH 파트 OK
AND       K00408	// W20-3 RH 작업완료 없음
AND=      0 D018508	// W20-3 RH 차종
LOAD      M00417	// W20-3 RH 차종이상
AND NOT   M00405	// W20 RH 이상해제
OR LOAD
AND       F0009A
OUT       M00417	// W20-3 RH 차종이상
; L44
LOAD      F0009A
LOAD      M00418	// W20 RH 이상
AND NOT   M00405	// W20 RH 이상해제
OR LOAD
OUT       M00418	// W20 RH 이상
; L46
LOAD      F0009A
LOAD      M00419	// W20 RH 이상
AND NOT   M00405	// W20 RH 이상해제
OR LOAD
OUT       M00419	// W20 RH 이상
; L48
LOAD      F0009A
LOAD      M0041A	// W20 RH 용접로봇 이상
AND NOT   M00405	// W20 RH 이상해제
OR LOAD
OUT       M0041A	// W20 RH 용접로봇 이상

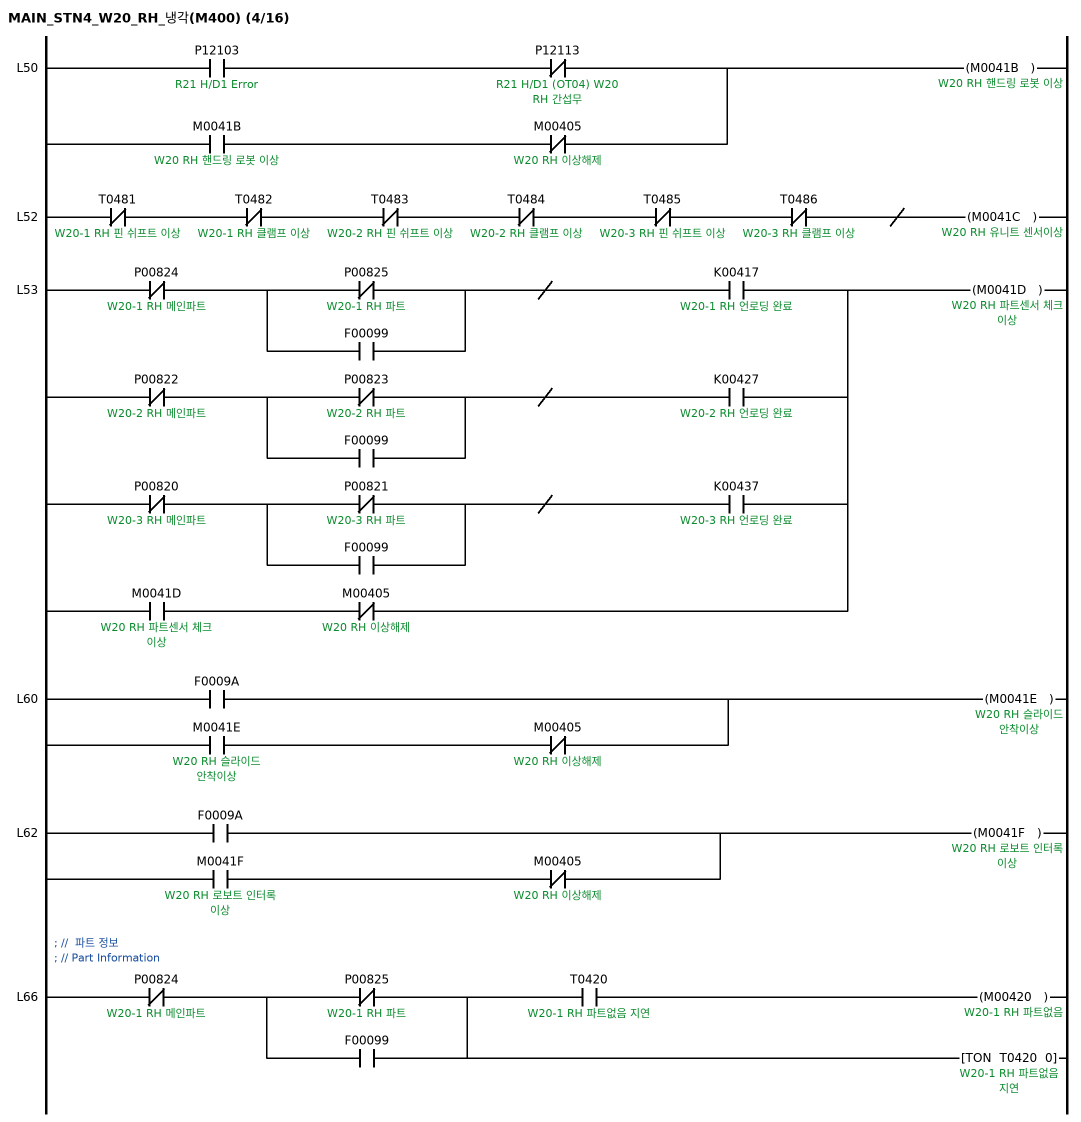
; L50
LOAD      P12103	// R21 H/D1 Error
AND NOT   P12113	// R21 H/D1 (OT04) W20 RH 간섭무
LOAD      M0041B	// W20 RH 핸드링 로봇 이상
AND NOT   M00405	// W20 RH 이상해제
OR LOAD
OUT       M0041B	// W20 RH 핸드링 로봇 이상
; L52
LOAD NOT  T0481	// W20-1 RH 핀 쉬프트 이상
AND NOT   T0482	// W20-1 RH 클램프 이상
AND NOT   T0483	// W20-2 RH 핀 쉬프트 이상
AND NOT   T0484	// W20-2 RH 클램프 이상
AND NOT   T0485	// W20-3 RH 핀 쉬프트 이상
AND NOT   T0486	// W20-3 RH 클램프 이상
NOT
OUT       M0041C	// W20 RH 유니트 센서이상
; L53
LOAD NOT  P00824	// W20-1 RH 메인파트
LOAD NOT  P00825	// W20-1 RH 파트
OR        F00099
AND LOAD
NOT
AND       K00417	// W20-1 RH 언로딩 완료
LOAD NOT  P00822	// W20-2 RH 메인파트
LOAD NOT  P00823	// W20-2 RH 파트
OR        F00099
AND LOAD
NOT
AND       K00427	// W20-2 RH 언로딩 완료
OR LOAD
LOAD NOT  P00820	// W20-3 RH 메인파트
LOAD NOT  P00821	// W20-3 RH 파트
OR        F00099
AND LOAD
NOT
AND       K00437	// W20-3 RH 언로딩 완료
OR LOAD
LOAD      M0041D	// W20 RH 파트센서 체크 이상
AND NOT   M00405	// W20 RH 이상해제
OR LOAD
OUT       M0041D	// W20 RH 파트센서 체크 이상
; L60
LOAD      F0009A
LOAD      M0041E	// W20 RH 슬라이드 안착이상
AND NOT   M00405	// W20 RH 이상해제
OR LOAD
OUT       M0041E	// W20 RH 슬라이드 안착이상
; L62
LOAD      F0009A
LOAD      M0041F	// W20 RH 로보트 인터록 이상
AND NOT   M00405	// W20 RH 이상해제
OR LOAD
OUT       M0041F	// W20 RH 로보트 인터록 이상
//   //  파트 정보
//   // Part Information
; L66
LOAD NOT  P00824	// W20-1 RH 메인파트
LOAD NOT  P00825	// W20-1 RH 파트
OR        F00099
AND LOAD
MPUSH
AND       T0420	// W20-1 RH 파트없음 지연
OUT       M00420	// W20-1 RH 파트없음
MPOP
TON       T0420 0	// W20-1 RH 파트없음 지연

